# B&R Automation Studio project AGV
Automation Studio 4.7.3.93 SP

## Configuration CP1586

CPU X20CP1586, AutomationRuntime B4.91, Build 4.1.2, Vc V4.72.3

### Task classes (Cpu.sw)
```
Cyclic#1 (cycle 5000 us, tolerance 5000 us):
  motorCtrl <- ros_topics_typ.motorCtrl.prg
Binaries: FWRules, TCData, udbdef, User, iomap, Role, arconfig, asfw, ashwac, sysconf, ashwd, target, components
Libraries: ExOS, ExDeploy, ExData, runtime, sys_lib, FileIO, AsIOTime, ArEventLog, AsTCP, ros_topics, ROS, operator, astime, AsIecCon, brsystem, MTTypes, standard, MTFilter, MTBasics
```

### Hardware
```
X20CP1586 : X20CP1586 v1.9.0.0
  Connector IF2:
    ActivateDevice = 1
    Mode = Manual
    InternetAddress = 192.168.87.212
    SubnetMask = 255.255.255.0
  ConfigurationID = AGV_CP1586
  IdleTaskClass = 3
  TaskClassIdleTime = 2000
  Cyclic1Duration = 5000
  Cyclic1Tolerance = 5000
  Cyclic2Duration = 1000
  FileDevice1
  FileDeviceName1 = USER
  FileDevicePath1 = USER_PATH
  ActivateOpcUa = 1
  OpcUaInformationModels_PV_Version = 1
```

### target.exostarget - X20CP1586/exosTechnology/target.exostarget
```
Element gTarget_0 (Type=exostarget)
  General:
    ConnectionIP = 192.168.87.128
    Logging:
      LogLevel = Debug
      LogFilters:
        LogFilterUser = On
        LogFilterSystem = On
        LogFilterVerbose = On
      LogDestination = Volatile
    Deployment = On
      MaxRestarts = 10
    DataConnection = On
      ConnectionType = TCPIP
      TimeSynchronization:
        TimeConnection:
          TimePort = 49001
        PrecisionUsec = 1000
        GuardTimeSec = 36
        DeviationPerHourUsec = 100000
      DataConnectionLogging:
        LogConnection:
          LogPort = 49002
          LogShmPath = exos_log
        LogCycleTimeMsec = 50
  Components:
    ComponentsGeneral:
      ComponentsHeartbeatMsec = 500
      ComponentsTimeoutSec = 2
      ComponentsTaskClass = 2
      ComponentsCycleTimeMsec = 10
    Component[0]:
      ComponentConfigurationLink = gros_topics_typ_0
      DataModels:
        Instance[0]:
          InstanceName = ros_topics_typ_0
          InstanceConnection:
            InstancePort = 49003
            InstanceShmPath = ros_topics_typ_0
  ComponentDataConnection:
    Version = 2.0.0-1
    ErrorHandling = Target
    RestartEvent = Target
    StartupTimeout = 5
    Predefined:
      Files:
        File[0]:
          FileName = ufw-exos-data
          ChangeEvent = Ignore
        File[1]:
          FileName = exos-data-ports-allow.sh
          ChangeEvent = Restart
        File[2]:
          FileName = exos-data.conf
          ChangeEvent = Restart
        File[3]:
          FileName = exos-data_2.0.0-1_amd64.deb
          ChangeEvent = Reinstall
        File[4]:
          FileName = exos-data-eth_2.0.0-1_amd64.deb
          ChangeEvent = Reinstall
        File[5]:
          FileName = exos-data-remove.sh
          ChangeEvent = Ignore
        File[6]:
          FileName = run_server.sh
          ChangeEvent = Ignore
        File[7]:
          FileName = setup_build_environment.sh
          ChangeEvent = Ignore
        File[8]:
          FileName = libzmq5_4.2.1-4+deb9u2_amd64.deb
          ChangeEvent = Reinstall
        File[9]:
          FileName = libpgm-5.2-0_5.2.122~dfsg-2_amd64.deb
          ChangeEvent = Reinstall
        File[10]:
          FileName = libsodium18_1.0.11-2_amd64.deb
          ChangeEvent = Reinstall
      Services:
        Service[0]:
          Type = Install
          Command = dpkg -i *.deb
          WorkingDirectory
        Service[1]:
          Type = Remove
          Command = dpkg --purge exos-data
          WorkingDirectory
        Service[2]:
          Type = Remove
          Command = dpkg --purge exos-data-eth
          WorkingDirectory
        Service[3]:
          Type = Remove
          Command = sh exos-data-remove.sh
          WorkingDirectory
        Service[4]:
          Type = Startup
          Command = cp exos-data.conf /etc/exos-data.conf
          WorkingDirectory
        Service[5]:
          Type = Startup
          Command = cp ufw-exos-data /etc/ufw/applications.d/ufw-exos-data
          WorkingDirectory
        Service[6]:
          Type = Startup
          Command = sh exos-data-ports-allow.sh
          WorkingDirectory
        Service[7]:
          Type = Runtime
          Command = /usr/bin/exos_mr
          WorkingDirectory
  Simulation:
    SimConnectionIP = 192.168.87.128
    SimDeployment = On
    SimDataConnection = On
      SimConnectionType = TCPIP
      SimTimeSynchronization:
        SimPrecisionUsec = 5000
        SimGuardTimeSec = 30
    SimComponentsGeneral:
      SimComponentsHeartbeatMsec = 1000
      SimComponentsTimeoutSec = 75
```

## Configuration Config1

CPU X90CP174.48-00, AutomationRuntime C4.72, Build 4.1.2, Vc V4.72.0

### Task classes (Cpu.sw)
```
Cyclic#1 (cycle 5000 us, tolerance 0 us):
  motorCtrl <- motorCtrl.prg
Binaries: udbdef, FWRules, TCData, iomap, ashwac, Role, sysconf, arconfig, asfw, User, ashwd
Libraries: MTBasics, brsystem, MTTypes, sys_lib, runtime, asieccon, astime, MTFilter, ROS, standard
```

### Hardware
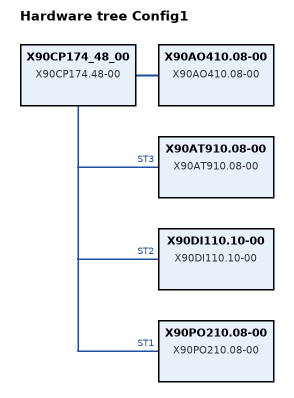
```
X90AO410.08-00 : X90AO410.08-00 v1.1.0.0  [ST -> X90CP174_48_00.ST4]
X90AT910.08-00 : X90AT910.08-00 v1.0.2.0  [ST -> X90CP174_48_00.ST3]
X90CP174_48_00 : X90CP174.48-00 v1.2.2.0  [X1 -> X1.SL]
  Module X1 (Type=X1, Virtual=true, Version=1.2.2.0)
    Connection (Connector=SL, TargetModule=X90CP174_48_00, TargetConnector=X1)
    ChannelConfig01 = 42
    DigitalFilterPin01 = 0
    ChannelConfig02 = 42
    DigitalFilterPin02 = 0
    ChannelConfig03 = 42
    DigitalFilterPin03 = 0
    ChannelConfig04 = 42
    DigitalFilterPin04 = 0
    IN1_CounterFunction01 = 3
    IN1_CounterFunction02 = 3
    ChannelConfig33 = 15
    PWMSource33 = 1
    PWMSyncPeriod33 = 125
    ChannelConfig34 = 20
    ChannelConfig35 = 20
    ChannelConfig36 = 20  // Configuration and impedance of pin X1.A.J1  
    ChannelConfig37 = 16
    ChannelConfig38 = 20  // Configuration and impedance of pin X1.A.L1  (6A)
    ChannelConfig39 = 20  // Configuration and impedance of pin X1.A.M2 (6A)
    ChannelConfig40 = 20
    ChannelConfig41 = 15
    PWMSource41 = 1
    PWMSyncPeriod41 = 125
    PWMDisplacement41 = 62
    ChannelConfig42 = 20
    ChannelConfig43 = 20  // Configuration and impedance of pin X1.B.H1  (6A)
    ChannelConfig44 = 20  // Configuration and impedance of pin X1.B.H3  (6A)
    ChannelConfig45 = 16  // Configuration and impedance of pin X1.B.G4  (6A)
    ChannelConfig46 = 20
    ChannelConfig47 = 20
    ChannelConfig48 = 20
  Connector IF2:
    ActivateDevice = 1
    Mode = Manual
    InternetAddress = 192.168.87.230
    SubnetMask = 255.255.255.0
  ConfigurationID = AGV_Config1
  EnableUsbRemoteInstall = 1
  EnableCfRemoteInstall = 1
  Cyclic1Duration = 5000
  Cyclic1Tolerance = 0
  Cyclic2Duration = 20000
  Cyclic2Tolerance = 20000
  Cyclic3Duration = 50000
  Cyclic3Tolerance = 50000
  Cyclic4Duration = 100000
  Cyclic4Tolerance = 100000
  Cyclic5Duration = 200000
  Cyclic5Tolerance = 200000
  Cyclic6Duration = 500000
  Cyclic6Tolerance = 500000
  Cyclic7Duration = 1000000
  Cyclic7Tolerance = 1000000
  Cyclic8Duration = 10000
  Cyclic8Tolerance = 30000000
  ActivateOpcUa = 1
  OpcUaInformationModels_PV_Version = 2
X90DI110.10-00 : X90DI110.10-00 v1.0.1.0  [ST -> X90CP174_48_00.ST2]
X90PO210.08-00 : X90PO210.08-00 v1.2.0.0  [ST -> X90CP174_48_00.ST1]
```

### IoMap.iom - X90CP174_48_00/IoMap.iom
```iecst
VAR_CONFIG
	::motorCtrl:localVariables[0].hw.output.pwm AT %QW."X1".PWMOutput33;
	::motorCtrl:localVariables[0].hw.input.encoder AT %IW."X1".Encoder01;
	::motorCtrl:localVariables[0].hw.input.current[0] AT %IW."X1".Current33;
	::motorCtrl:localVariables[0].hw.input.current[1] AT %IW."X1".Current34;
	::motorCtrl:localVariables[0].hw.input.current[2] AT %IW."X1".Current35;
	::motorCtrl:localVariables[0].hw.input.current[3] AT %IW."X1".Current36;
	::motorCtrl:localVariables[0].hw.input.overload AT %IX."X1".OverloadDigitalOutput33;
	::motorCtrl:localVariables[0].hw.output.clear AT %QX."X1".OverloadClear33;
	::motorCtrl:localVariables[1].hw.input.encoder AT %IW."X1".Encoder02;
	::motorCtrl:localVariables[1].hw.output.pwm AT %QW."X1".PWMOutput37;
	::motorCtrl:localVariables[0].hw.input.current[4] AT %IW."X1".Current37;
	::motorCtrl:localVariables[0].hw.input.current[6] AT %IW."X1".Current39;
	::motorCtrl:localVariables[1].hw.input.nettime AT %ID."X90CP174_48_00".SystemTime;
	::motorCtrl:localVariables[0].hw.input.nettime AT %ID."X90CP174_48_00".SystemTime;
	::motorCtrl:localVariables[0].hw.input.current[5] AT %IW."X1".Current38;
	::motorCtrl:localVariables[0].hw.input.current[7] AT %IW."X1".Current40;
	::motorCtrl:localVariables[1].hw.output.pwm AT %QW."X1".PWMOutput41;
	::motorCtrl:localVariables[1].hw.output.clear AT %QX."X1".OverloadClear41;
	::motorCtrl:localVariables[1].hw.input.current[0] AT %IW."X1".Current41;
	::motorCtrl:localVariables[1].hw.input.overload  AT %IX."X1".OverloadDigitalOutput41;
	::motorCtrl:localVariables[1].hw.input.current[1]  AT %IW."X1".Current42;
	::motorCtrl:localVariables[1].hw.input.current[2]  AT %IW."X1".Current43;
	::motorCtrl:localVariables[1].hw.input.current[3]  AT %IW."X1".Current44;
	::motorCtrl:localVariables[1].hw.input.current[4]  AT %IW."X1".Current45;
	::motorCtrl:localVariables[1].hw.input.current[5]  AT %IW."X1".Current46;
	::motorCtrl:localVariables[1].hw.input.current[6]  AT %IW."X1".Current47;
	::motorCtrl:localVariables[1].hw.input.current[7]  AT %IW."X1".Current48;
END_VAR
```

### components.exoscomponent - X90CP174_48_00/exosTechnology/components.exoscomponent
```
Element gros_topics_typ_0 (Type=exoscomponent)
  PackageSelection = Logical\ros_topics_typ\ros_topics_typ.exospkg
  ErrorHandling = Component
  RestartEvent = Component
  StartupTimeout = 0
  Predefined:
    Files:
      File[0]:
        FileName = Linux\ros_topics_typ.py
        ChangeEvent = Restart
      File[1]:
        FileName = Linux\exos-comp-ros_topics_typ_1.0.0_amd64.deb
        ChangeEvent = Reinstall
    Services:
      Service[0]:
        Type = Install
        Command = dpkg -i exos-comp-ros_topics_typ_1.0.0_amd64.deb
        WorkingDirectory
      Service[1]:
        Type = Remove
        Command = dpkg --purge exos-comp-ros_topics_typ
        WorkingDirectory
      Service[2]:
        Type = Startup
        Command = cp ros_topics_typ.py /home/user/brdkAGV_linux/ros_ws/src/motor_control_exos/motor_control_exos/motor_control_exos.py
        WorkingDirectory
Element gWaterTank_0 (Type=exoscomponent)
  PackageSelection = Logical\WaterTank\WaterTank.exospkg
  ErrorHandling = Component
  RestartEvent = Component
  StartupTimeout = 0
  Predefined:
    Files:
      File[0]:
        FileName = Linux\watertank.py
        ChangeEvent = Restart
      File[1]:
        FileName = Linux\exos-comp-watertank_1.0.0_amd64.deb
        ChangeEvent = Reinstall
    Services:
      Service[0]:
        Type = Install
        Command = dpkg -i exos-comp-watertank_1.0.0_amd64.deb
        WorkingDirectory
      Service[1]:
        Type = Remove
        Command = dpkg --purge exos-comp-watertank
        WorkingDirectory
      Service[2]:
        Type = Startup
        Command = cp watertank.py /home/user/watertank
        WorkingDirectory
      Service[3]:
        Type = Runtime
        Command = python3 watertank.py
        WorkingDirectory = /home/user/watertank
```

### target.exostarget - X90CP174_48_00/exosTechnology/target.exostarget
```
Element gTarget_0 (Type=exostarget)
  General:
    ConnectionIP = 192.168.87.128
    Logging:
      LogLevel = Debug
      LogFilters:
        LogFilterUser = On
        LogFilterSystem = On
        LogFilterVerbose = On
      LogDestination = Volatile
    Deployment = On
      MaxRestarts = 10
    DataConnection = On
      ConnectionType = TCPIP
      TimeSynchronization:
        TimeConnection:
          TimePort = 49001
        PrecisionUsec = 5000
        GuardTimeSec = 180
        DeviationPerHourUsec = 100000
      DataConnectionLogging:
        LogConnection:
          LogPort = 49002
          LogShmPath = exos_log
        LogCycleTimeMsec = 50
  Components:
    ComponentsGeneral:
      ComponentsHeartbeatMsec = 500
      ComponentsTimeoutSec = 2
      ComponentsTaskClass = 2
      ComponentsCycleTimeMsec = 10
    Component[0]:
      ComponentConfigurationLink = gros_topics_typ_0
      DataModels:
        Instance[0]:
          InstanceName = ros_topics_typ_0
          InstanceConnection:
            InstancePort = 49003
            InstanceShmPath = ros_topics_typ_0
    Component[1]:
      ComponentConfigurationLink = gWaterTank_0
      DataModels:
        Instance[0]:
          InstanceName = WaterTank_0
          InstanceConnection:
            InstancePort = 49004
            InstanceShmPath = WaterTank_0
  ComponentDataConnection:
    Version = 2.1.0-1
    ErrorHandling = Target
    RestartEvent = Target
    StartupTimeout = 5
    Predefined:
      Files:
        File[0]:
          FileName = ufw-exos-data
          ChangeEvent = Ignore
        File[1]:
          FileName = exos-data-ufw-profile.sh
          ChangeEvent = Ignore
        File[2]:
          FileName = exos-data-ports-allow.sh
          ChangeEvent = Restart
        File[3]:
          FileName = exos-data.conf
          ChangeEvent = Restart
        File[4]:
          FileName = exos-data_2.1.0-1_amd64.deb
          ChangeEvent = Reinstall
        File[5]:
          FileName = exos-data-eth_2.1.0-1_amd64.deb
          ChangeEvent = Reinstall
        File[6]:
          FileName = exos-data-remove.sh
          ChangeEvent = Ignore
        File[7]:
          FileName = run_server.sh
          ChangeEvent = Ignore
        File[8]:
          FileName = setup_build_environment.sh
          ChangeEvent = Ignore
        File[9]:
          FileName = libzmq5_4.2.1-4+deb9u2_amd64.deb
          ChangeEvent = Reinstall
        File[10]:
          FileName = libpgm-5.2-0_5.2.122~dfsg-2_amd64.deb
          ChangeEvent = Reinstall
        File[11]:
          FileName = libsodium18_1.0.11-2_amd64.deb
          ChangeEvent = Reinstall
      Services:
        Service[0]:
          Type = Install
          Command = dpkg -i *.deb
          WorkingDirectory
        Service[1]:
          Type = Remove
          Command = dpkg --purge exos-data
          WorkingDirectory
        Service[2]:
          Type = Remove
          Command = dpkg --purge exos-data-eth
          WorkingDirectory
        Service[3]:
          Type = Remove
          Command = sh exos-data-remove.sh
          WorkingDirectory
        Service[4]:
          Type = Startup
          Command = cp exos-data.conf /etc/exos-data.conf
          WorkingDirectory
        Service[5]:
          Type = Startup
          Command = sh exos-data-ufw-profile.sh
          WorkingDirectory
        Service[6]:
          Type = Startup
          Command = sh exos-data-ports-allow.sh
          WorkingDirectory
        Service[7]:
          Type = Runtime
          Command = /usr/bin/exos_mr
          WorkingDirectory
  Simulation:
    SimConnectionIP = 192.168.87.128
    SimDeployment = On
    SimDataConnection = On
      SimConnectionType = TCPIP
      SimTimeSynchronization:
        SimPrecisionUsec = 10000
        SimGuardTimeSec = 30
    SimComponentsGeneral:
      SimComponentsHeartbeatMsec = 1000
      SimComponentsTimeoutSec = 75
```

## Logical view

Binary libraries used (declarations not repeated): operator, runtime, astime, AsIecCon, MTBasics 5.06.0, brsystem, MTTypes, sys_lib, MTFilter 5.06.0, standard, AsIOTime, ExOS 2.01.0

### Package Logical/Libraries - Global libraries

### Library Logical/Libraries/ROS (ANSIC)

#### Types.typ - Exported data types
```iecst
TYPE
	ros_topic_point_typ : 	STRUCT  (*this expresses velocity in free space broken into its linear and angular parts.*)
		y : LREAL;
		z : LREAL;
		x : LREAL;
	END_STRUCT;
	ros_topic_vector3_typ : 	STRUCT  (*this expresses velocity in free space broken into its linear and angular parts.*)
		y : LREAL;
		z : LREAL;
		x : LREAL;
	END_STRUCT;
	ros_topic_twist_typ : 	STRUCT  (*This expresses velocity in free space broken into its linear and angular parts.*)
		angular : ros_topic_vector3_typ;
		linear : ros_topic_vector3_typ;
	END_STRUCT;
	ros_topic_twistCor_typ : 	STRUCT  (*This expresses velocity in free space with uncertainty.*)
		twist : ros_topic_twist_typ;
		covariance : ARRAY[0..63]OF LREAL; (*Row-major representation of the 6x6 covariance matrix
The orientation parameters use a fixed-axis representation. In order, the parameters are:
 (x, y, z, rotation about X axis, rotation about Y axis, rotation about Z axis)*)
	END_STRUCT;
	ros_topic_quaternion_typ : 	STRUCT  (*This represents an orientation in free space in quaternion form.*)
		y : LREAL;
		z : LREAL;
		w : LREAL;
		x : LREAL;
	END_STRUCT;
	ros_topic_odemety_point_typ : 	STRUCT  (*This contains the position of a point in free space*)
		y : LREAL;
		z : LREAL;
		x : LREAL;
	END_STRUCT;
	ros_topic_pose_typ : 	STRUCT  (*A representation of pose in free space, composed of position and orientation. *)
		position : ros_topic_point_typ;
		orientation : ros_topic_quaternion_typ;
	END_STRUCT;
	ros_topic_poseCor_typ : 	STRUCT  (*This represents a pose in free space with uncertainty.*)
		pose : ros_topic_pose_typ;
		covariance : ARRAY[0..63]OF LREAL; (*Row-major representation of the 6x6 covariance matrix
The orientation parameters use a fixed-axis representation. In order, the parameters are:
 (x, y, z, rotation about X axis, rotation about Y axis, rotation about Z axis)*)
	END_STRUCT;
	ros_topic_time_typ : 	STRUCT
		nsec : UDINT;
		sec : UDINT;
	END_STRUCT;
	ros_topic_header_typ : 	STRUCT
		stamp : ros_topic_time_typ;
		seq : UDINT;
		frame_id : STRING[20];
	END_STRUCT;
	ros_topic_odemety_typ : 	STRUCT
		pose : ros_topic_poseCor_typ;
		twist : ros_topic_twistCor_typ;
		header : ros_topic_header_typ;
	END_STRUCT;
END_TYPE
```

#### ROS.fun - Exported functions and function blocks
```iecst
{REDUND_ERROR} FUNCTION normalizeAngle : LREAL (*TODO: Add your comment here*) (*$GROUP=User,$CAT=User,$GROUPICON=User.png,$CATICON=User.png*)
	VAR_INPUT
		angle : LREAL;
	END_VAR
END_FUNCTION
```

#### normalizeAngle.c
```c
#include <bur/plctypes.h>
#ifdef __cplusplus
	extern "C"
	{
#endif
	#include "ROS.h"
#ifdef __cplusplus
	};
#endif

#define M_PI 3.14159265358979323846

/* TODO: Add your comment here */
double normalizeAngle(double angle)
{

	if( angle > M_PI){
		angle -= 2.0 * M_PI;
	}
	if(angle < -M_PI){
		angle += 2.0 * M_PI;
	}

	return angle;
}
```

### Program Logical/motorCtrl (IEC)

#### Main.st - Init, cyclic, exit code
```iecst
PROGRAM _INIT
	(* Insert code here *)
	FOR i:=0 TO i < 2 BY 1 DO
		setupPointers;

		this.PID.Enable := TRUE;
		this.PID.MinOut := -100;
		this.PID.MaxOut := 100;
		this.PID.PIDParameters.DerivativeTime := 0.00228000456;
		this.PID.PIDParameters.Gain := 78;
		this.PID.PIDParameters.IntegrationTime := 0.02500019;
		this.PID.PIDParameters.FilterTime := 0.000228000456;

		this.PID.Update := TRUE;

		this.PIDCurrent.Enable := TRUE;
		this.PIDCurrent.MinOut := 0;
		this.PIDCurrent.MaxOut := 100;
		this.PIDCurrent.PIDParameters.DerivativeTime := 10;
		this.PIDCurrent.PIDParameters.Gain := 1;
		this.PIDCurrent.PIDParameters.IntegrationTime := 10;
		this.PIDCurrent.PIDParameters.FilterTime := 20;
		this.PIDCurrent.Update := TRUE;
		this.PIDCurrent.SetValue := 8;

		this.filterSpeed.Enable := TRUE;
		this.filterSpeed.WindowLength := 100;
		this.filterSpeed.Update := TRUE;

		this.filterCurrent.Enable := TRUE;
		this.filterCurrent.WindowLength := 3;
		this.filterCurrent.Update := TRUE;

		this.accLimiter.Enable := TRUE;
		this.accLimiter.MaxNegSlewRate := 1;
		this.accLimiter.MaxPosSlewRate := 1;
		this.accLimiter.MaxOut := 2;
		this.accLimiter.MinOut := -2;
		this.accLimiter.Update := TRUE;

		this.PIDtune.SetValue:= 1.0;
		this.PIDtune.MinOut:= 0.0;
		this.PIDtune.MaxOut:= 100.0;
		this.PIDtune.Update := TRUE;

		this.lowPass.Enable := TRUE;
		this.lowPass.CutOffFrequency := 10;
		this.lowPass.Order := 1;
		this.lowPass.Update := TRUE;

		this.encoderOld := this.hw.input.encoder;
		this.timeOld := this.hw.input.nettime;

		this.ton_overcurrent.PT := T#1s;

	END_FOR

END_PROGRAM

PROGRAM _CYCLIC
	(* Insert code here *)

	ros.topics.twist.linear.x := MAX(MIN(ros.topics.twist.linear.x,ros.topics.config.maxSpeed),ros.topics.config.minSpeed);

	IF localVariables[0].hmi.output.overload OR localVariables[1].hmi.output.overload  THEN
		localVariables[0].PID.SetValue := 0;
		localVariables[1].PID.SetValue := 0;
	ELSE
		localVariables[0].PID.SetValue := LREAL_TO_REAL(ros.topics.twist.linear.x + ros.topics.twist.angular.z * ros.topics.config.baseWidth / 2.0) * ros.currentLimiter;  // m/s
		localVariables[1].PID.SetValue := LREAL_TO_REAL(ros.topics.twist.linear.x - ros.topics.twist.angular.z * ros.topics.config.baseWidth / 2.0) * ros.currentLimiter;
	END_IF

	FOR i:=0 TO 1 BY 1 DO
		setupPointers;

		hmi.output.overload := FALSE;

		hmi.output.currentTotal := 0;

		FOR k:=0 TO 7 DO

			hmi.output.current[k] := INT_TO_REAL(hw.input.current[k])*10.0/32767.0;
			hmi.output.currentTotal := hmi.output.currentTotal + hmi.output.current[k];
		END_FOR

		hmi.output.currentTotal := hmi.output.currentTotal /2.0;

		IF this.filterCurrent.UpdateDone THEN
			this.filterSpeed.Update := FALSE;
		END_IF

		this.filterCurrent(In := hmi.output.currentTotal);

		IF this.PIDCurrent.UpdateDone THEN
			this.PIDCurrent.Update := FALSE;
		END_IF

		this.PIDCurrent(ActValue := this.filterCurrent.Out);

		this.currentLimiter := 1;//this.PIDCurrent.Out/100;

		hmi.output.overload := hw.input.overload;

		this.ton_overcurrent(IN := hmi.output.overload);
		IF this.ton_overcurrent.Q THEN
			this.hmi.input.clear := TRUE;
		END_IF

		hw.output.clear := hmi.input.clear;

		IF NOT hmi.output.overload THEN
			hmi.input.clear := FALSE;
		END_IF

		this.diffTime := DINT_TO_LREAL(hw.input.nettime -this.timeOld);
		IF this.diffTime < -100000.0 THEN
			this.diffTime := this.diffTime + 2*2147483647;
		END_IF
		this.diffTime := this.diffTime /1000.0;
		this.timeOld := hw.input.nettime;

		this.diffEncoder := INT_TO_LREAL(hw.input.encoder)-INT_TO_LREAL(this.encoderOld);

		this.encoderOld := hw.input.encoder;

		IF this.diffEncoder > 32727 THEN

			this.diffEncoder := this.diffEncoder - 2*32767;

		ELSIF this.diffEncoder < -32727 THEN

			this.diffEncoder := this.diffEncoder + 2*32767;

		END_IF

		hmi.output.ticks := hmi.output.ticks + this.diffEncoder;
		hmi.output.distance := hmi.output.ticks / UDINT_TO_LREAL(config.ppm);

		IF hmi.input.resetDistance THEN
			hmi.input.resetDistance := FALSE;
			hmi.output.ticks := 0;
			hmi.output.distance := 0;
		END_IF

		this.distance 	:= this.diffEncoder/UDINT_TO_LREAL(config.ppm);

		this.lowPass.In := LREAL_TO_REAL(this.distance);
		this.lowPass();

		this.speed 		:= this.distance * 1000/this.diffTime;

		IF this.filterSpeed.UpdateDone THEN
			this.filterSpeed.Update := FALSE;
		END_IF

		this.filterSpeed(In := LREAL_TO_REAL(this.speed));

		IF this.accLimiter.UpdateDone THEN
			this.accLimiter.Update := FALSE;
		END_IF

		this.accLimiter(In := this.PID.SetValue);

		IF this.PID.UpdateDone THEN
			this.PID.Update := FALSE;
		END_IF

		this.PID.ActValue := LREAL_TO_REAL(this.speed);
		this.PID.SetValue := this.accLimiter.Out;
		// PID TUNE

		IF hmi.input.tune THEN
			this.PIDtune.Enable := TRUE;
		END_IF

		this.PIDtune.ActValue := LREAL_TO_REAL(this.speed);

		IF this.PIDtune.TuningDone THEN
			this.PIDtune.Start := FALSE;
			this.PID.IntegrationPartPresetValue := this.PIDtune.Out;
			this.PID.SetIntegrationPart := TRUE;
		ELSIF this.PIDtune.Active AND NOT this.PIDtune.Update THEN
			//	this.PIDtune.Start := TRUE;
		END_IF

		IF this.PIDtune.UpdateDone THEN
			this.PIDtune.Update := FALSE;
		END_IF

		(* call function block *)
		this.PID();
		this.PIDtune();

		this.PID.SetIntegrationPart := FALSE;

		IF hmi.input.tune THEN
			hw.output.pwm := REAL_TO_INT(this.PIDtune.Out*327.67);
		ELSE
			hw.output.pwm := REAL_TO_INT(this.PID.Out*327.67);
		END_IF

	END_FOR

	ros.currentLimiter := MIN(localVariables[0].currentLimiter,localVariables[1].currentLimiter);

	ros.diffDist := localVariables[1].distance-localVariables[0].distance;
	ros.diffLowpassDist := localVariables[1].lowPass.Out-localVariables[0].lowPass.Out;

	ros.dist := (localVariables[1].distance+localVariables[0].distance)/2;

	IF localVariables[0].diffEncoder = localVariables[1].diffEncoder THEN
		ros.d_theta := 0.0;
		ros.cur_x := ros.cur_x + ros.dist * COS(ros.cur_theta);
		ros.cur_y := ros.cur_y + ros.dist * SIN(ros.cur_theta);
	ELSE
		ros.d_theta := (localVariables[1].distance - localVariables[0].distance) / ros.topics.config.baseWidth;
		ros.dist := (localVariables[1].distance+localVariables[0].distance)/2;
		ros.r := ros.dist / ros.d_theta;
		ros.cur_x := ros.cur_x + ros.r * (SIN(ros.d_theta + ros.cur_theta) - SIN(ros.cur_theta));
		ros.cur_y := ros.cur_y - ros.r * (COS(ros.d_theta + ros.cur_theta) - COS(ros.cur_theta));
		ros.cur_theta := normalizeAngle(ros.cur_theta + ros.d_theta);
	END_IF

	ros.vel_x := ros.dist * (1000.0/localVariables[0].diffTime);
	ros.vel_theta := ros.d_theta * (1000.0/localVariables[0].diffTime);

	// set ros data
	ros.topics.odemetry.pose.pose.position.x 	:= ros.cur_x;
	ros.topics.odemetry.pose.pose.position.y	:= ros.cur_y;
	ros.topics.odemetry.pose.pose.orientation.z	:= ros.cur_theta;

	ros.topics.odemetry.twist.twist.linear.x  	:= ros.vel_x;
	ros.topics.odemetry.twist.twist.angular.z 	:= ros.vel_theta;

	setupWatchPointers;

END_PROGRAM

PROGRAM _EXIT
	(* Insert code here *)

END_PROGRAM
```

#### Types.typ - Local data types
```iecst
TYPE
	ros_config_typ : 	STRUCT
		maxSpeed : LREAL := 2;
		minSpeed : LREAL := -2;
		baseWidth : LREAL := 0.53;
	END_STRUCT;
	ros_topics_typ : 	STRUCT
		odemetry : ros_topic_odemety_typ;
		twist : ros_topic_twist_typ;
		config : ros_config_typ;
	END_STRUCT;
	ros_typ : 	STRUCT
		vel_theta : LREAL;
		vel_x : LREAL;
		r : LREAL;
		cur_theta : LREAL;
		dist : LREAL;
		cur_y : LREAL;
		cur_x : LREAL;
		d_theta : LREAL;
		topics : ros_topics_typ;
		diffLowpassDist : REAL;
		diffDist : LREAL;
		currentLimiter : REAL;
	END_STRUCT;
	local_typ : 	STRUCT
		hw : hw_typ;
		hmi : hmi_typ;
		speed : LREAL;
		encoderOld : INT;
		accLimiter : MTBasicsLimiter;
		PIDCurrent : MTBasicsPID;
		PID : MTBasicsPID;
		distance : LREAL;
		diffEncoder : LREAL;
		filterCurrent : MTFilterMovingAverage;
		filterSpeed : MTFilterMovingAverage;
		diffTime : LREAL;
		timeOld : DINT;
		PIDtune : MTBasicsOscillationTuning;
		lowPass : MTFilterLowPass;
		ton_overcurrent : TON;
		currentLimiter : REAL;
	END_STRUCT;
	hw_typ : 	STRUCT
		input : hw_input_typ;
		output : hw_output_typ;
	END_STRUCT;
	hw_output_typ : 	STRUCT
		pwm : INT;
		clear : BOOL;
	END_STRUCT;
	hw_input_typ : 	STRUCT
		encoder : INT;
		overload : BOOL;
		current : ARRAY[0..7]OF INT;
		nettime : DINT;
	END_STRUCT;
	hmi_typ : 	STRUCT
		config : config_typ;
		output : hmi_output_typ;
		input : hmi_input_typ;
	END_STRUCT;
	hmi_output_typ : 	STRUCT
		current : ARRAY[0..7]OF REAL;
		overload : BOOL;
		distance : LREAL;
		ticks : LREAL;
		currentTotal : REAL;
	END_STRUCT;
	hmi_input_typ : 	STRUCT
		clear : BOOL;
		tune : BOOL;
		resetDistance : BOOL;
	END_STRUCT;
	config_typ : 	STRUCT
		ppm : UDINT := 105860;
		maxCurrent : REAL := 8;
	END_STRUCT;
	common_typ : 	STRUCT
	END_STRUCT;
END_TYPE
```

#### Variables.var - Local variables
```iecst
VAR
	ros : ros_typ;
	config : REFERENCE TO config_typ;
	hmi : REFERENCE TO hmi_typ;
	hw : REFERENCE TO hw_typ;
	this : REFERENCE TO local_typ;
	localVariables : ARRAY[0..1] OF local_typ;
	watchIdx : USINT;
	k : USINT;
	i : USINT;
END_VAR
```

- ros_topics_typ.exospkg (not shown)

### libros_topics_typ.c - ros_topics_typ static library wrapper source
```c
#include <string.h>
#define EXOS_ASSERT_LOG &logger
#include "exos_log.h"
#include "libros_topics_typ.h"

#define SUCCESS(_format_, ...) exos_log_success(&logger, EXOS_LOG_TYPE_USER, _format_, ##__VA_ARGS__);
#define INFO(_format_, ...) exos_log_info(&logger, EXOS_LOG_TYPE_USER, _format_, ##__VA_ARGS__);
#define VERBOSE(_format_, ...) exos_log_debug(&logger, EXOS_LOG_TYPE_USER + EXOS_LOG_TYPE_VERBOSE, _format_, ##__VA_ARGS__);
#define ERROR(_format_, ...) exos_log_error(&logger, _format_, ##__VA_ARGS__);

static exos_log_handle_t logger;

typedef struct libros_topics_typHandle
{
    libros_topics_typ_t ext_ros_topics_typ_datamodel;
    exos_datamodel_handle_t ros_topics_typ_datamodel;

    exos_dataset_handle_t odemetry_dataset;
    exos_dataset_handle_t twist_dataset;
    exos_dataset_handle_t config_dataset;
} libros_topics_typHandle_t;

static libros_topics_typHandle_t h_ros_topics_typ;

static void libros_topics_typ_datasetEvent(exos_dataset_handle_t *dataset, EXOS_DATASET_EVENT_TYPE event_type, void *info)
{
    switch (event_type)
    {
    case EXOS_DATASET_EVENT_UPDATED:
        VERBOSE("dataset %s updated! latency (us):%i", dataset->name, (exos_datamodel_get_nettime(dataset->datamodel) - dataset->nettime));
        //handle each subscription dataset separately
        if (0 == strcmp(dataset->name, "odemetry"))
        {
            //update the nettime
            h_ros_topics_typ.ext_ros_topics_typ_datamodel.odemetry.nettime = dataset->nettime;

            //trigger the callback if assigned
            if (NULL != h_ros_topics_typ.ext_ros_topics_typ_datamodel.odemetry.on_change)
            {
                h_ros_topics_typ.ext_ros_topics_typ_datamodel.odemetry.on_change();
            }
        }
        break;

    default:
        break;
    }
}

static void libros_topics_typ_datamodelEvent(exos_datamodel_handle_t *datamodel, const EXOS_DATAMODEL_EVENT_TYPE event_type, void *info)
{
    switch (event_type)
    {
    case EXOS_DATAMODEL_EVENT_CONNECTION_CHANGED:
        INFO("application changed state to %s", exos_get_state_string(datamodel->connection_state));

        h_ros_topics_typ.ext_ros_topics_typ_datamodel.is_connected = false;
        h_ros_topics_typ.ext_ros_topics_typ_datamodel.is_operational = false;
        switch (datamodel->connection_state)
        {
        case EXOS_STATE_DISCONNECTED:
            if (NULL != h_ros_topics_typ.ext_ros_topics_typ_datamodel.on_disconnected)
            {
                h_ros_topics_typ.ext_ros_topics_typ_datamodel.on_disconnected();
            }
            break;
        case EXOS_STATE_CONNECTED:
            h_ros_topics_typ.ext_ros_topics_typ_datamodel.is_connected = true;
            if (NULL != h_ros_topics_typ.ext_ros_topics_typ_datamodel.on_connected)
            {
                h_ros_topics_typ.ext_ros_topics_typ_datamodel.on_connected();
            }
            break;
        case EXOS_STATE_OPERATIONAL:
            h_ros_topics_typ.ext_ros_topics_typ_datamodel.is_connected = true;
            h_ros_topics_typ.ext_ros_topics_typ_datamodel.is_operational = true;
            if (NULL != h_ros_topics_typ.ext_ros_topics_typ_datamodel.on_operational)
            {
                h_ros_topics_typ.ext_ros_topics_typ_datamodel.on_operational();
            }
            SUCCESS("ros_topics_typ operational!");
            break;
        case EXOS_STATE_ABORTED:
            if (NULL != h_ros_topics_typ.ext_ros_topics_typ_datamodel.on_disconnected)
            {
                h_ros_topics_typ.ext_ros_topics_typ_datamodel.on_disconnected();
            }
            ERROR("application error %d (%s) occured", datamodel->error, exos_get_error_string(datamodel->error));
            break;
        }
        break;
    case EXOS_DATAMODEL_EVENT_SYNC_STATE_CHANGED:
        break;

    default:
        break;

    }
}

static void libros_topics_typ_publish_twist_dataset(void)
{
    exos_dataset_publish(&h_ros_topics_typ.twist_dataset);
}
static void libros_topics_typ_publish_config_dataset(void)
{
    exos_dataset_publish(&h_ros_topics_typ.config_dataset);
}

static void libros_topics_typ_connect(void)
{
    //connect the datamodel
    EXOS_ASSERT_OK(exos_datamodel_connect_ros_topics_typ(&(h_ros_topics_typ.ros_topics_typ_datamodel), libros_topics_typ_datamodelEvent));

    //connect datasets
    EXOS_ASSERT_OK(exos_dataset_connect(&(h_ros_topics_typ.odemetry_dataset), EXOS_DATASET_SUBSCRIBE, libros_topics_typ_datasetEvent));
    EXOS_ASSERT_OK(exos_dataset_connect(&(h_ros_topics_typ.twist_dataset), EXOS_DATASET_PUBLISH, libros_topics_typ_datasetEvent));
    EXOS_ASSERT_OK(exos_dataset_connect(&(h_ros_topics_typ.config_dataset), EXOS_DATASET_PUBLISH, libros_topics_typ_datasetEvent));
}
static void libros_topics_typ_disconnect(void)
{
    h_ros_topics_typ.ext_ros_topics_typ_datamodel.is_connected = false;
    h_ros_topics_typ.ext_ros_topics_typ_datamodel.is_operational = false;

    EXOS_ASSERT_OK(exos_datamodel_disconnect(&(h_ros_topics_typ.ros_topics_typ_datamodel)));
}

static void libros_topics_typ_set_operational(void)
{
    EXOS_ASSERT_OK(exos_datamodel_set_operational(&(h_ros_topics_typ.ros_topics_typ_datamodel)));
}

static void libros_topics_typ_process(void)
{
    EXOS_ASSERT_OK(exos_datamodel_process(&(h_ros_topics_typ.ros_topics_typ_datamodel)));
    exos_log_process(&logger);
}

static void libros_topics_typ_dispose(void)
{
    h_ros_topics_typ.ext_ros_topics_typ_datamodel.is_connected = false;
    h_ros_topics_typ.ext_ros_topics_typ_datamodel.is_operational = false;

    EXOS_ASSERT_OK(exos_datamodel_delete(&(h_ros_topics_typ.ros_topics_typ_datamodel)));
    exos_log_delete(&logger);
}

static int32_t libros_topics_typ_get_nettime(void)
{
    return exos_datamodel_get_nettime(&(h_ros_topics_typ.ros_topics_typ_datamodel));
}

static void libros_topics_typ_log_error(char* log_entry)
{
    exos_log_error(&logger, log_entry);
}

static void libros_topics_typ_log_warning(char* log_entry)
{
    exos_log_warning(&logger, EXOS_LOG_TYPE_USER, log_entry);
}

static void libros_topics_typ_log_success(char* log_entry)
{
    exos_log_success(&logger, EXOS_LOG_TYPE_USER, log_entry);
}

static void libros_topics_typ_log_info(char* log_entry)
{
    exos_log_info(&logger, EXOS_LOG_TYPE_USER, log_entry);
}

static void libros_topics_typ_log_debug(char* log_entry)
{
    exos_log_debug(&logger, EXOS_LOG_TYPE_USER, log_entry);
}

static void libros_topics_typ_log_verbose(char* log_entry)
{
    exos_log_warning(&logger, EXOS_LOG_TYPE_USER + EXOS_LOG_TYPE_VERBOSE, log_entry);
}

libros_topics_typ_t *libros_topics_typ_init(void)
{
    memset(&h_ros_topics_typ, 0, sizeof(h_ros_topics_typ));

    h_ros_topics_typ.ext_ros_topics_typ_datamodel.twist.publish = libros_topics_typ_publish_twist_dataset;
    h_ros_topics_typ.ext_ros_topics_typ_datamodel.config.publish = libros_topics_typ_publish_config_dataset;

    h_ros_topics_typ.ext_ros_topics_typ_datamodel.connect = libros_topics_typ_connect;
    h_ros_topics_typ.ext_ros_topics_typ_datamodel.disconnect = libros_topics_typ_disconnect;
    h_ros_topics_typ.ext_ros_topics_typ_datamodel.process = libros_topics_typ_process;
    h_ros_topics_typ.ext_ros_topics_typ_datamodel.set_operational = libros_topics_typ_set_operational;
    h_ros_topics_typ.ext_ros_topics_typ_datamodel.dispose = libros_topics_typ_dispose;
    h_ros_topics_typ.ext_ros_topics_typ_datamodel.get_nettime = libros_topics_typ_get_nettime;
    h_ros_topics_typ.ext_ros_topics_typ_datamodel.log.error = libros_topics_typ_log_error;
    h_ros_topics_typ.ext_ros_topics_typ_datamodel.log.warning = libros_topics_typ_log_warning;
    h_ros_topics_typ.ext_ros_topics_typ_datamodel.log.success = libros_topics_typ_log_success;
    h_ros_topics_typ.ext_ros_topics_typ_datamodel.log.info = libros_topics_typ_log_info;
    h_ros_topics_typ.ext_ros_topics_typ_datamodel.log.debug = libros_topics_typ_log_debug;
    h_ros_topics_typ.ext_ros_topics_typ_datamodel.log.verbose = libros_topics_typ_log_verbose;

    exos_log_init(&logger, "gros_topics_typ_0");

    SUCCESS("starting gros_topics_typ_0 application..");

    EXOS_ASSERT_OK(exos_datamodel_init(&h_ros_topics_typ.ros_topics_typ_datamodel, "ros_topics_typ_0", "gros_topics_typ_0"));

    //set the user_context to access custom data in the callbacks
    h_ros_topics_typ.ros_topics_typ_datamodel.user_context = NULL; //not used
    h_ros_topics_typ.ros_topics_typ_datamodel.user_tag = 0; //not used

    EXOS_ASSERT_OK(exos_dataset_init(&h_ros_topics_typ.odemetry_dataset, &h_ros_topics_typ.ros_topics_typ_datamodel, "odemetry", &h_ros_topics_typ.ext_ros_topics_typ_datamodel.odemetry.value, sizeof(h_ros_topics_typ.ext_ros_topics_typ_datamodel.odemetry.value)));
    h_ros_topics_typ.odemetry_dataset.user_context = NULL; //not used
    h_ros_topics_typ.odemetry_dataset.user_tag = 0; //not used

    EXOS_ASSERT_OK(exos_dataset_init(&h_ros_topics_typ.twist_dataset, &h_ros_topics_typ.ros_topics_typ_datamodel, "twist", &h_ros_topics_typ.ext_ros_topics_typ_datamodel.twist.value, sizeof(h_ros_topics_typ.ext_ros_topics_typ_datamodel.twist.value)));
    h_ros_topics_typ.twist_dataset.user_context = NULL; //not used
    h_ros_topics_typ.twist_dataset.user_tag = 0; //not used

    EXOS_ASSERT_OK(exos_dataset_init(&h_ros_topics_typ.config_dataset, &h_ros_topics_typ.ros_topics_typ_datamodel, "config", &h_ros_topics_typ.ext_ros_topics_typ_datamodel.config.value, sizeof(h_ros_topics_typ.ext_ros_topics_typ_datamodel.config.value)));
    h_ros_topics_typ.config_dataset.user_context = NULL; //not used
    h_ros_topics_typ.config_dataset.user_tag = 0; //not used

    return &(h_ros_topics_typ.ext_ros_topics_typ_datamodel);
}
```

### CMakeLists.txt - CMake build file script
```
cmake_minimum_required(VERSION 3.0)

project(ros_topics_typ)

set(CMAKE_BUILD_TYPE Debug)
find_package(SWIG REQUIRED)
include(${SWIG_USE_FILE})

# Load Python Libraries
# ---------------------
# a.) use Python 3
find_package(PythonLibs 3)
# b.) use Python 2.7 (  change the Runtime service command to 'python2' in the .exospkg file)
# - update the DEPENDS to python-dev
# find_package(PythonLibs 2)
# c.) use pyenv to manually install a version matching the Python version on the target distro https://realpython.com/intro-to-pyenv/
# set(PYTHON_INCLUDE_PATH ~/.pyenv/versions/3.9-dev/include/python3.9)
# set(PYTHON_LIBRARIES ~/.pyenv/versions/3.9-dev/lib/libpython3.9.so)

include_directories(${PYTHON_INCLUDE_PATH})

include_directories(${CMAKE_CURRENT_SOURCE_DIR})

set(CMAKE_SWIG_FLAGS "")

set(ROS_TOPICS_TYP_SOURCES
    libros_topics_typ.c
    libros_topics_typ.i
    exos_ros_topics_typ.c
    )

set_source_files_properties(${ROS_TOPICS_TYP_SOURCES} PROPERTIES CPLUSPLUS ON)

swig_add_module(libros_topics_typ python ${ROS_TOPICS_TYP_SOURCES})
swig_link_libraries(libros_topics_typ ${PYTHON_LIBRARIES} zmq exos-api)

set(ROS_TOPICS_TYP_MODULE_FILES
    build/_libros_topics_typ.so
    build/libros_topics_typ.py
    )

install(FILES ${ROS_TOPICS_TYP_MODULE_FILES} DESTINATION /home/user/ros_topics_typ)

set(CPACK_GENERATOR "DEB")
set(CPACK_PACKAGE_NAME exos-comp-ros_topics_typ)
set(CPACK_PACKAGE_DESCRIPTION_SUMMARY "ros_topics_typ summary")
set(CPACK_PACKAGE_DESCRIPTION "Some description")
set(CPACK_PACKAGE_VENDOR "Your Company")

set(CPACK_PACKAGE_VERSION_MAJOR 1)
set(CPACK_PACKAGE_VERSION_MINOR 0)
set(CPACK_PACKAGE_VERSION_PATCH 0)
set(CPACK_PACKAGE_FILE_NAME exos-comp-ros_topics_typ_1.0.0_amd64)
set(CPACK_DEBIAN_PACKAGE_MAINTAINER "Your Name")

set(CPACK_DEBIAN_PACKAGE_SHLIBDEPS ON)

include(CPack)
```

- ros_topics_typ.py - Main python script (not shown)

- _libros_topics_typ.so - ros_topics_typ SWIG library (binary file, 581832 bytes)
- ros_topics_typ1.py - Main python script (not shown)

### Program Logical/ros_topics_typ/motorCtrl

#### ros_topics_typ.var
```iecst
VAR
	ros_topics_typInit_0 : ros_topics_typInit;
	ros_topics_typCyclic_0 : ros_topics_typCyclic;
	ros_topics_typExit_0 : ros_topics_typExit;
	ExComponentInfo_0 : ExComponentInfo;
	ExDatamodelInfo_0 : ExDatamodelInfo;
	ros : ros_typ;
	config : REFERENCE TO config_typ;
	hmi : REFERENCE TO hmi_typ;
	hw : REFERENCE TO hw_typ;
	this : REFERENCE TO local_typ;
	localVariables : ARRAY[0..1] OF local_typ;
	watchIdx : USINT;
	k : USINT;
	i : USINT;
END_VAR
```

#### ros_topics_typ.st
```iecst
PROGRAM _INIT

	ros_topics_typInit_0();

	(* Insert code here *)
	FOR i:=0 TO i < 2 BY 1 DO
		setupPointers;

		this.PID.Enable := TRUE;
		this.PID.MinOut := -100;
		this.PID.MaxOut := 100;
		this.PID.PIDParameters.DerivativeTime := 0.00228000456;
		this.PID.PIDParameters.Gain := 78;
		this.PID.PIDParameters.IntegrationTime := 0.02500019;
		this.PID.PIDParameters.FilterTime := 0.000228000456;

		this.PID.Update := TRUE;

		this.PIDCurrent.Enable := TRUE;
		this.PIDCurrent.MinOut := 0;
		this.PIDCurrent.MaxOut := 100;
		this.PIDCurrent.PIDParameters.DerivativeTime := 10;
		this.PIDCurrent.PIDParameters.Gain := 1;
		this.PIDCurrent.PIDParameters.IntegrationTime := 10;
		this.PIDCurrent.PIDParameters.FilterTime := 20;
		this.PIDCurrent.Update := TRUE;
		this.PIDCurrent.SetValue := 8;

		this.filterSpeed.Enable := TRUE;
		this.filterSpeed.WindowLength := 100;
		this.filterSpeed.Update := TRUE;

		this.filterCurrent.Enable := TRUE;
		this.filterCurrent.WindowLength := 3;
		this.filterCurrent.Update := TRUE;

		this.accLimiter.Enable := TRUE;
		this.accLimiter.MaxNegSlewRate := 1;
		this.accLimiter.MaxPosSlewRate := 1;
		this.accLimiter.MaxOut := 2;
		this.accLimiter.MinOut := -2;
		this.accLimiter.Update := TRUE;

		this.PIDtune.SetValue:= 1.0;
		this.PIDtune.MinOut:= 0.0;
		this.PIDtune.MaxOut:= 100.0;
		this.PIDtune.Update := TRUE;

		this.lowPass.Enable := TRUE;
		this.lowPass.CutOffFrequency := 10;
		this.lowPass.Order := 1;
		this.lowPass.Update := TRUE;

		this.encoderOld := this.hw.input.encoder;
		this.timeOld := this.hw.input.nettime;

		this.ton_overcurrent.PT := T#1s;

	END_FOR

END_PROGRAM

PROGRAM _CYCLIC
    //--------------- ex OS ----------------
    //Auto connect:
	ros_topics_typCyclic_0.Enable := ExComponentInfo_0.Operational; // Component has been deployed and started up successfully

	//Auto connect when deployment is off and manually started in GPOS:
	//ros_topics_typCyclic_0.Enable := TRUE;
	ros_topics_typCyclic_0.Start := ros_topics_typCyclic_0.Connected;

	ros_topics_typCyclic_0(Handle := ros_topics_typInit_0.Handle, pros_topics_typ := ADR(ros.topics));

	ExComponentInfo_0(ExTargetLink := ADR(gTarget_0), ExComponentLink := ADR(gros_topics_typ_0), Enable := TRUE);

	ExDatamodelInfo_0(ExTargetLink := ADR(gTarget_0), Enable := TRUE, InstanceName := 'ros_topics_typ_0');
	//--------------- ex OS done ----------------
	ExSyncInfo_0(ExTargetLink := ADR(gTarget_0), Enable := TRUE);

	ros.topics.twist.linear.x := MAX(MIN(ros.topics.twist.linear.x,ros.topics.config.maxSpeed),ros.topics.config.minSpeed);

	IF localVariables[0].hmi.output.overload OR localVariables[1].hmi.output.overload OR NOT ros_topics_typCyclic_0.Operational THEN
		localVariables[0].PID.SetValue := 0;
		localVariables[1].PID.SetValue := 0;
	ELSE
		localVariables[0].PID.SetValue := LREAL_TO_REAL(ros.topics.twist.linear.x + ros.topics.twist.angular.z * ros.topics.config.baseWidth / 2.0) * ros.currentLimiter;  // m/s
		localVariables[1].PID.SetValue := LREAL_TO_REAL(ros.topics.twist.linear.x - ros.topics.twist.angular.z * ros.topics.config.baseWidth / 2.0) * ros.currentLimiter;
	END_IF

	FOR i:=0 TO 1 BY 1 DO
		setupPointers;

		hmi.output.overload := FALSE;

		hmi.output.currentTotal := 0;

		FOR k:=0 TO 7 DO

			hmi.output.current[k] := INT_TO_REAL(hw.input.current[k])*10.0/32767.0;
			hmi.output.currentTotal := hmi.output.currentTotal + hmi.output.current[k];
		END_FOR

		hmi.output.currentTotal := hmi.output.currentTotal /2.0;

		IF this.filterCurrent.UpdateDone THEN
			this.filterSpeed.Update := FALSE;
		END_IF

		this.filterCurrent(In := hmi.output.currentTotal);

		IF this.PIDCurrent.UpdateDone THEN
			this.PIDCurrent.Update := FALSE;
		END_IF

		this.PIDCurrent(ActValue := this.filterCurrent.Out);

		this.currentLimiter := 1;//this.PIDCurrent.Out/100;

		hmi.output.overload := hw.input.overload;

		this.ton_overcurrent(IN := hmi.output.overload);
		IF this.ton_overcurrent.Q THEN
			this.hmi.input.clear := TRUE;
		END_IF

		hw.output.clear := hmi.input.clear;

		IF NOT hmi.output.overload THEN
			hmi.input.clear := FALSE;
		END_IF

		this.diffTime := DINT_TO_LREAL(hw.input.nettime -this.timeOld);
		IF this.diffTime < -100000.0 THEN
			this.diffTime := this.diffTime + 2*2147483647;
		END_IF
		this.diffTime := this.diffTime /1000.0;
		this.timeOld := hw.input.nettime;

		this.diffEncoder := INT_TO_LREAL(hw.input.encoder)-INT_TO_LREAL(this.encoderOld);

		this.encoderOld := hw.input.encoder;

		IF this.diffEncoder > 32727 THEN

			this.diffEncoder := this.diffEncoder - 2*32767;

		ELSIF this.diffEncoder < -32727 THEN

			this.diffEncoder := this.diffEncoder + 2*32767;

		END_IF

		hmi.output.ticks := hmi.output.ticks + this.diffEncoder;
		hmi.output.distance := hmi.output.ticks / UDINT_TO_LREAL(config.ppm);

		IF hmi.input.resetDistance THEN
			hmi.input.resetDistance := FALSE;
			hmi.output.ticks := 0;
			hmi.output.distance := 0;
		END_IF

		this.distance 	:= this.diffEncoder/UDINT_TO_LREAL(config.ppm);

		this.lowPass.In := LREAL_TO_REAL(this.distance);
		this.lowPass();

		this.speed 		:= this.distance * 1000/this.diffTime;

		IF this.filterSpeed.UpdateDone THEN
			this.filterSpeed.Update := FALSE;
		END_IF

		this.filterSpeed(In := LREAL_TO_REAL(this.speed));

		IF this.accLimiter.UpdateDone THEN
			this.accLimiter.Update := FALSE;
		END_IF

		this.accLimiter(In := this.PID.SetValue);

		IF this.PID.UpdateDone THEN
			this.PID.Update := FALSE;
		END_IF

		this.PID.ActValue := LREAL_TO_REAL(this.speed);
		this.PID.SetValue := this.accLimiter.Out;
		// PID TUNE

		IF hmi.input.tune THEN
			this.PIDtune.Enable := TRUE;
		END_IF

		this.PIDtune.ActValue := LREAL_TO_REAL(this.speed);

		IF this.PIDtune.TuningDone THEN
			this.PIDtune.Start := FALSE;
			this.PID.IntegrationPartPresetValue := this.PIDtune.Out;
			this.PID.SetIntegrationPart := TRUE;
		ELSIF this.PIDtune.Active AND NOT this.PIDtune.Update THEN
			//	this.PIDtune.Start := TRUE;
		END_IF

		IF this.PIDtune.UpdateDone THEN
			this.PIDtune.Update := FALSE;
		END_IF

		(* call function block *)
		this.PID();
		this.PIDtune();

		this.PID.SetIntegrationPart := FALSE;

		IF hmi.input.tune THEN
			hw.output.pwm := REAL_TO_INT(this.PIDtune.Out*327.67);
		ELSE
			hw.output.pwm := REAL_TO_INT(this.PID.Out*327.67);
		END_IF

	END_FOR

	ros.currentLimiter := MIN(localVariables[0].currentLimiter,localVariables[1].currentLimiter);

	ros.diffDist := localVariables[1].distance-localVariables[0].distance;
	ros.diffLowpassDist := localVariables[1].lowPass.Out-localVariables[0].lowPass.Out;

	ros.dist := (localVariables[1].distance+localVariables[0].distance)/2;

	IF localVariables[0].diffEncoder = localVariables[1].diffEncoder THEN
		ros.d_theta := 0.0;
		ros.cur_x := ros.cur_x + ros.dist * COS(ros.cur_theta);
		ros.cur_y := ros.cur_y + ros.dist * SIN(ros.cur_theta);
	ELSE
		ros.d_theta := (localVariables[1].distance - localVariables[0].distance) / ros.topics.config.baseWidth;
		ros.dist := (localVariables[1].distance+localVariables[0].distance)/2;
		ros.r := ros.dist / ros.d_theta;
		ros.cur_x := ros.cur_x + ros.r * (SIN(ros.d_theta + ros.cur_theta) - SIN(ros.cur_theta));
		ros.cur_y := ros.cur_y - ros.r * (COS(ros.d_theta + ros.cur_theta) - COS(ros.cur_theta));
		ros.cur_theta := normalizeAngle(ros.cur_theta + ros.d_theta);
	END_IF

	ros.vel_x := ros.dist * (1000.0/localVariables[0].diffTime);
	ros.vel_theta := ros.d_theta * (1000.0/localVariables[0].diffTime);

	// set ros data
	ros.topics.odemetry.pose.pose.position.x 	:= ros.cur_x;
	ros.topics.odemetry.pose.pose.position.y	:= ros.cur_y;
	ros.topics.odemetry.pose.pose.orientation.z	:= ros.cur_theta;

	ros.topics.odemetry.twist.twist.linear.x  	:= ros.vel_x;
	ros.topics.odemetry.twist.twist.angular.z 	:= ros.vel_theta;

	setupWatchPointers;

END_PROGRAM

PROGRAM _EXIT

	ros_topics_typExit_0(Handle := ros_topics_typInit_0.Handle);

END_PROGRAM
```

#### setupPointers.st
```iecst
ACTION setupPointers:

	this ACCESS ADR(localVariables[i]);
	config ACCESS ADR(localVariables[i].hmi.config);
	hw ACCESS ADR(localVariables[i].hw);
	hmi ACCESS ADR(localVariables[i].hmi);

END_ACTION

ACTION setupWatchPointers:

	i := watchIdx;
	this ACCESS ADR(localVariables[i]);
	config ACCESS ADR(localVariables[i].hmi.config);
	hw ACCESS ADR(localVariables[i].hw);
	hmi ACCESS ADR(localVariables[i].hmi);

END_ACTION
```

### ros_topics_typ.var
```iecst
VAR
    ros_topics_typInit_0 : ros_topics_typInit;
    ros_topics_typCyclic_0 : ros_topics_typCyclic;
    ros_topics_typExit_0 : ros_topics_typExit;
    ros_topics_typ_0 : ros_topics_typ;
    ExComponentInfo_0 : ExComponentInfo;
    ExDatamodelInfo_0 : ExDatamodelInfo;
END_VAR
```

### Program Logical/ros_topics_typ - Copy/motorCtrl (IEC) - ros_topics_typ application

#### motorCtrl.typ - Local data types
```iecst
TYPE
	ros_typ : 	STRUCT
		vel_theta : LREAL;
		vel_x : LREAL;
		r : LREAL;
		cur_theta : LREAL;
		dist : LREAL;
		cur_y : LREAL;
		cur_x : LREAL;
		d_theta : LREAL;
		topics : ros_topics_typ;
		diffLowpassDist : REAL;
		diffDist : LREAL;
		currentLimiter : REAL;
	END_STRUCT;
	local_typ : 	STRUCT
		hw : hw_typ;
		hmi : hmi_typ;
		speed : LREAL;
		encoderOld : INT;
		accLimiter : MTBasicsLimiter;
		PIDCurrent : MTBasicsPID;
		PID : MTBasicsPID;
		distance : LREAL;
		diffEncoder : LREAL;
		filterCurrent : MTFilterMovingAverage;
		filterSpeed : MTFilterMovingAverage;
		diffTime : LREAL;
		timeOld : DINT;
		PIDtune : MTBasicsOscillationTuning;
		lowPass : MTFilterLowPass;
		ton_overcurrent : TON;
		currentLimiter : REAL;
	END_STRUCT;
	hw_typ : 	STRUCT
		input : hw_input_typ;
		output : hw_output_typ;
	END_STRUCT;
	hw_output_typ : 	STRUCT
		pwm : INT;
		clear : BOOL;
	END_STRUCT;
	hw_input_typ : 	STRUCT
		encoder : INT;
		overload : BOOL;
		current : ARRAY[0..7]OF INT;
		nettime : DINT;
	END_STRUCT;
	hmi_typ : 	STRUCT
		config : config_typ;
		output : hmi_output_typ;
		input : hmi_input_typ;
	END_STRUCT;
	hmi_output_typ : 	STRUCT
		current : ARRAY[0..7]OF REAL;
		overload : BOOL;
		distance : LREAL;
		ticks : LREAL;
		currentTotal : REAL;
	END_STRUCT;
	hmi_input_typ : 	STRUCT
		clear : BOOL;
		tune : BOOL;
		resetDistance : BOOL;
	END_STRUCT;
	config_typ : 	STRUCT
		ppm : UDINT := 105860;
		maxCurrent : REAL := 8;
	END_STRUCT;
	common_typ : 	STRUCT
	END_STRUCT;
END_TYPE
```

#### ros_topics_typ.var - ros_topics_typ variable declaration
```iecst
VAR
	ros_topics_typInit_0 : ros_topics_typInit;
	ros_topics_typCyclic_0 : ros_topics_typCyclic;
	ros_topics_typExit_0 : ros_topics_typExit;
	ExComponentInfo_0 : ExComponentInfo;
	ExSyncInfo_0 : ExSyncInfo;
	ExDatamodelInfo_0 : ExDatamodelInfo;
	ros : ros_typ;
	config : REFERENCE TO config_typ;
	hmi : REFERENCE TO hmi_typ;
	hw : REFERENCE TO hw_typ;
	this : REFERENCE TO local_typ;
	localVariables : ARRAY[0..1] OF local_typ;
	watchIdx : USINT;
	k : USINT;
	i : USINT;
END_VAR
```

### Library Logical/ros_topics_typ - Copy/ros_topics (ANSIC) - ros_topics_typ exOS library
Depends on: ExData

#### exos_ros_topics_typ.c - Generated datamodel source for ros_topics_typ
```c
/*Automatically generated c file from ros_topics_typ.typ*/

#include "exos_ros_topics_typ.h"

const char config_ros_topics_typ[] = "{\"name\":\"struct\",\"attributes\":{\"name\":\"<NAME>\",\"dataType\":\"ros_topics_typ\",\"info\":\"<infoId0>\"},\"children\":[{\"name\":\"struct\",\"attributes\":{\"name\":\"odemetry\",\"dataType\":\"ros_topic_odemety_typ\",\"comment\":\"PUB\",\"info\":\"<infoId1>\"},\"children\":[{\"name\":\"struct\",\"attributes\":{\"name\":\"pose\",\"dataType\":\"ros_topic_poseCor_typ\",\"info\":\"<infoId2>\"},\"children\":[{\"name\":\"struct\",\"attributes\":{\"name\":\"pose\",\"dataType\":\"ros_topic_pose_typ\",\"info\":\"<infoId3>\"},\"children\":[{\"name\":\"struct\",\"attributes\":{\"name\":\"position\",\"dataType\":\"ros_topic_point_typ\",\"info\":\"<infoId4>\"},\"children\":[{\"name\":\"variable\",\"attributes\":{\"name\":\"y\",\"dataType\":\"LREAL\",\"info\":\"<infoId5>\"}},{\"name\":\"variable\",\"attributes\":{\"name\":\"z\",\"dataType\":\"LREAL\",\"info\":\"<infoId6>\"}},{\"name\":\"variable\",\"attributes\":{\"name\":\"x\",\"dataType\":\"LREAL\",\"info\":\"<infoId7>\"}}]},{\"name\":\"struct\",\"attributes\":{\"name\":\"orientation\",\"dataType\":\"ros_topic_quaternion_typ\",\"info\":\"<infoId8>\"},\"children\":[{\"name\":\"variable\",\"attributes\":{\"name\":\"y\",\"dataType\":\"LREAL\",\"info\":\"<infoId9>\"}},{\"name\":\"variable\",\"attributes\":{\"name\":\"z\",\"dataType\":\"LREAL\",\"info\":\"<infoId10>\"}},{\"name\":\"variable\",\"attributes\":{\"name\":\"w\",\"dataType\":\"LREAL\",\"info\":\"<infoId11>\"}},{\"name\":\"variable\",\"attributes\":{\"name\":\"x\",\"dataType\":\"LREAL\",\"info\":\"<infoId12>\"}}]}]}]},{\"name\":\"struct\",\"attributes\":{\"name\":\"twist\",\"dataType\":\"ros_topic_twistCor_typ\",\"info\":\"<infoId13>\"},\"children\":[{\"name\":\"struct\",\"attributes\":{\"name\":\"twist\",\"dataType\":\"ros_topic_twist_typ\",\"info\":\"<infoId14>\"},\"children\":[{\"name\":\"struct\",\"attributes\":{\"name\":\"angular\",\"dataType\":\"ros_topic_vector3_typ\",\"info\":\"<infoId15>\"},\"children\":[{\"name\":\"variable\",\"attributes\":{\"name\":\"y\",\"dataType\":\"LREAL\",\"info\":\"<infoId16>\"}},{\"name\":\"variable\",\"attributes\":{\"name\":\"z\",\"dataType\":\"LREAL\",\"info\":\"<infoId17>\"}},{\"name\":\"variable\",\"attributes\":{\"name\":\"x\",\"dataType\":\"LREAL\",\"info\":\"<infoId18>\"}}]},{\"name\":\"struct\",\"attributes\":{\"name\":\"linear\",\"dataType\":\"ros_topic_vector3_typ\",\"info\":\"<infoId19>\"},\"children\":[{\"name\":\"variable\",\"attributes\":{\"name\":\"y\",\"dataType\":\"LREAL\",\"info\":\"<infoId20>\"}},{\"name\":\"variable\",\"attributes\":{\"name\":\"z\",\"dataType\":\"LREAL\",\"info\":\"<infoId21>\"}},{\"name\":\"variable\",\"attributes\":{\"name\":\"x\",\"dataType\":\"LREAL\",\"info\":\"<infoId22>\"}}]}]}]},{\"name\":\"struct\",\"attributes\":{\"name\":\"header\",\"dataType\":\"ros_topic_header_typ\",\"info\":\"<infoId23>\"},\"children\":[{\"name\":\"struct\",\"attributes\":{\"name\":\"stamp\",\"dataType\":\"ros_topic_time_typ\",\"info\":\"<infoId24>\"},\"children\":[{\"name\":\"variable\",\"attributes\":{\"name\":\"nsec\",\"dataType\":\"UDINT\",\"info\":\"<infoId25>\"}},{\"name\":\"variable\",\"attributes\":{\"name\":\"sec\",\"dataType\":\"UDINT\",\"info\":\"<infoId26>\"}}]},{\"name\":\"variable\",\"attributes\":{\"name\":\"seq\",\"dataType\":\"UDINT\",\"info\":\"<infoId27>\"}},{\"name\":\"variable\",\"attributes\":{\"name\":\"frame_id\",\"dataType\":\"STRING\",\"stringLength\":21,\"info\":\"<infoId28>\"}}]}]},{\"name\":\"struct\",\"attributes\":{\"name\":\"twist\",\"dataType\":\"ros_topic_twist_typ\",\"comment\":\"SUB\",\"info\":\"<infoId29>\"},\"children\":[{\"name\":\"struct\",\"attributes\":{\"name\":\"angular\",\"dataType\":\"ros_topic_vector3_typ\",\"info\":\"<infoId30>\"},\"children\":[{\"name\":\"variable\",\"attributes\":{\"name\":\"y\",\"dataType\":\"LREAL\",\"info\":\"<infoId31>\"}},{\"name\":\"variable\",\"attributes\":{\"name\":\"z\",\"dataType\":\"LREAL\",\"info\":\"<infoId32>\"}},{\"name\":\"variable\",\"attributes\":{\"name\":\"x\",\"dataType\":\"LREAL\",\"info\":\"<infoId33>\"}}]},{\"name\":\"struct\",\"attributes\":{\"name\":\"linear\",\"dataType\":\"ros_topic_vector3_typ\",\"info\":\"<infoId34>\"},\"children\":[{\"name\":\"variable\",\"attributes\":{\"name\":\"y\",\"dataType\":\"LREAL\",\"info\":\"<infoId35>\"}},{\"name\":\"variable\",\"attributes\":{\"name\":\"z\",\"dataType\":\"LREAL\",\"info\":\"<infoId36>\"}},{\"name\":\"variable\",\"attributes\":{\"name\":\"x\",\"dataType\":\"LREAL\",\"info\":\"<infoId37>\"}}]}]},{\"name\":\"struct\",\"attributes\":{\"name\":\"config\",\"dataType\":\"ros_config_typ\",\"comment\":\"SUB\",\"info\":\"<infoId38>\"},\"children\":[{\"name\":\"variable\",\"attributes\":{\"name\":\"maxSpeed\",\"dataType\":\"LREAL\",\"info\":\"<infoId39>\"}},{\"name\":\"variable\",\"attributes\":{\"name\":\"minSpeed\",\"dataType\":\"LREAL\",\"info\":\"<infoId40>\"}},{\"name\":\"variable\",\"attributes\":{\"name\":\"baseWidth\",\"dataType\":\"LREAL\",\"info\":\"<infoId41>\"}}]}]}";

/*Connect the ros_topics_typ datamodel to the server*/
EXOS_ERROR_CODE exos_datamodel_connect_ros_topics_typ(exos_datamodel_handle_t *datamodel, exos_datamodel_event_cb datamodel_event_callback)
{
    ros_topics_typ data;
    exos_dataset_info_t datasets[] = {
        {EXOS_DATASET_BROWSE_NAME_INIT,{}},
        {EXOS_DATASET_BROWSE_NAME(odemetry),{}},
        {EXOS_DATASET_BROWSE_NAME(odemetry.pose),{}},
        {EXOS_DATASET_BROWSE_NAME(odemetry.pose.pose),{}},
        {EXOS_DATASET_BROWSE_NAME(odemetry.pose.pose.position),{}},
        {EXOS_DATASET_BROWSE_NAME(odemetry.pose.pose.position.y),{}},
        {EXOS_DATASET_BROWSE_NAME(odemetry.pose.pose.position.z),{}},
        {EXOS_DATASET_BROWSE_NAME(odemetry.pose.pose.position.x),{}},
        {EXOS_DATASET_BROWSE_NAME(odemetry.pose.pose.orientation),{}},
        {EXOS_DATASET_BROWSE_NAME(odemetry.pose.pose.orientation.y),{}},
        {EXOS_DATASET_BROWSE_NAME(odemetry.pose.pose.orientation.z),{}},
        {EXOS_DATASET_BROWSE_NAME(odemetry.pose.pose.orientation.w),{}},
        {EXOS_DATASET_BROWSE_NAME(odemetry.pose.pose.orientation.x),{}},
        {EXOS_DATASET_BROWSE_NAME(odemetry.twist),{}},
        {EXOS_DATASET_BROWSE_NAME(odemetry.twist.twist),{}},
        {EXOS_DATASET_BROWSE_NAME(odemetry.twist.twist.angular),{}},
        {EXOS_DATASET_BROWSE_NAME(odemetry.twist.twist.angular.y),{}},
        {EXOS_DATASET_BROWSE_NAME(odemetry.twist.twist.angular.z),{}},
        {EXOS_DATASET_BROWSE_NAME(odemetry.twist.twist.angular.x),{}},
        {EXOS_DATASET_BROWSE_NAME(odemetry.twist.twist.linear),{}},
        {EXOS_DATASET_BROWSE_NAME(odemetry.twist.twist.linear.y),{}},
        {EXOS_DATASET_BROWSE_NAME(odemetry.twist.twist.linear.z),{}},
        {EXOS_DATASET_BROWSE_NAME(odemetry.twist.twist.linear.x),{}},
        {EXOS_DATASET_BROWSE_NAME(odemetry.header),{}},
        {EXOS_DATASET_BROWSE_NAME(odemetry.header.stamp),{}},
        {EXOS_DATASET_BROWSE_NAME(odemetry.header.stamp.nsec),{}},
        {EXOS_DATASET_BROWSE_NAME(odemetry.header.stamp.sec),{}},
        {EXOS_DATASET_BROWSE_NAME(odemetry.header.seq),{}},
        {EXOS_DATASET_BROWSE_NAME(odemetry.header.frame_id),{}},
        {EXOS_DATASET_BROWSE_NAME(twist),{}},
        {EXOS_DATASET_BROWSE_NAME(twist.angular),{}},
        {EXOS_DATASET_BROWSE_NAME(twist.angular.y),{}},
        {EXOS_DATASET_BROWSE_NAME(twist.angular.z),{}},
        {EXOS_DATASET_BROWSE_NAME(twist.angular.x),{}},
        {EXOS_DATASET_BROWSE_NAME(twist.linear),{}},
        {EXOS_DATASET_BROWSE_NAME(twist.linear.y),{}},
        {EXOS_DATASET_BROWSE_NAME(twist.linear.z),{}},
        {EXOS_DATASET_BROWSE_NAME(twist.linear.x),{}},
        {EXOS_DATASET_BROWSE_NAME(config),{}},
        {EXOS_DATASET_BROWSE_NAME(config.maxSpeed),{}},
        {EXOS_DATASET_BROWSE_NAME(config.minSpeed),{}},
        {EXOS_DATASET_BROWSE_NAME(config.baseWidth),{}}
    };

    exos_datamodel_calc_dataset_info(datasets, sizeof(datasets));

    return exos_datamodel_connect(datamodel, config_ros_topics_typ, datasets, sizeof(datasets), datamodel_event_callback);
}
```

### Package Logical/ros_topics_typ - Copy/Linux - ros_topics_typ Linux resources

### exos_ros_topics_typ.h
```c
/*Automatically generated header file from ros_topics_typ.typ*/

#ifndef _EXOS_COMP_ROS_TOPICS_TYP_H_
#define _EXOS_COMP_ROS_TOPICS_TYP_H_

#include "exos_api.h"

#if defined(_SG4)
#include <ros_topics.h>
#else
#include <stddef.h>
#include <stdint.h>
#include <stdbool.h>

typedef struct ros_config_typ
{
    double maxSpeed;
    double minSpeed;
    double baseWidth;

} ros_config_typ;

typedef struct ros_topic_vector3_typ
{
    double y;
    double z;
    double x;

} ros_topic_vector3_typ;

typedef struct ros_topic_twist_typ
{
    struct ros_topic_vector3_typ angular;
    struct ros_topic_vector3_typ linear;

} ros_topic_twist_typ;

typedef struct ros_topic_time_typ
{
    uint32_t nsec;
    uint32_t sec;

} ros_topic_time_typ;

typedef struct ros_topic_header_typ
{
    struct ros_topic_time_typ stamp;
    uint32_t seq;
    char frame_id[21];

} ros_topic_header_typ;

typedef struct ros_topic_twistCor_typ
{
    struct ros_topic_twist_typ twist;

} ros_topic_twistCor_typ;

typedef struct ros_topic_quaternion_typ
{
    double y;
    double z;
    double w;
    double x;

} ros_topic_quaternion_typ;

typedef struct ros_topic_point_typ
{
    double y;
    double z;
    double x;

} ros_topic_point_typ;

typedef struct ros_topic_pose_typ
{
    struct ros_topic_point_typ position;
    struct ros_topic_quaternion_typ orientation;

} ros_topic_pose_typ;

typedef struct ros_topic_poseCor_typ
{
    struct ros_topic_pose_typ pose;

} ros_topic_poseCor_typ;

typedef struct ros_topic_odemety_typ
{
    struct ros_topic_poseCor_typ pose;
    struct ros_topic_twistCor_typ twist;
    struct ros_topic_header_typ header;

} ros_topic_odemety_typ;

typedef struct ros_topics_typ
{
    struct ros_topic_odemety_typ odemetry; //PUB
    struct ros_topic_twist_typ twist; //SUB
    struct ros_config_typ config; //SUB

} ros_topics_typ;

#endif // _SG4

EXOS_ERROR_CODE exos_datamodel_connect_ros_topics_typ(exos_datamodel_handle_t *datamodel, exos_datamodel_event_cb datamodel_event_callback);

#endif // _EXOS_COMP_ROS_TOPICS_TYP_H_
```

- libros_topics_typ.py (not shown)

- ros_topics_typ.py (not shown)

### ros_topics.typ
```iecst
TYPE
	ros_topic_point_typ : 	STRUCT  (*this expresses velocity in free space broken into its linear and angular parts.*)
		y : LREAL;
		z : LREAL;
		x : LREAL;
	END_STRUCT;
	ros_topic_vector3_typ : 	STRUCT  (*this expresses velocity in free space broken into its linear and angular parts.*)
		y : LREAL;
		z : LREAL;
		x : LREAL;
	END_STRUCT;
	ros_topic_twist_typ : 	STRUCT  (*This expresses velocity in free space broken into its linear and angular parts.*)
		angular : ros_topic_vector3_typ;
		linear : ros_topic_vector3_typ;
	END_STRUCT;
	ros_topic_twistCor_typ : 	STRUCT  (*This expresses velocity in free space with uncertainty.*)
		twist : ros_topic_twist_typ;
	END_STRUCT;
	ros_topic_quaternion_typ : 	STRUCT  (*This represents an orientation in free space in quaternion form.*)
		y : LREAL;
		z : LREAL;
		w : LREAL;
		x : LREAL;
	END_STRUCT;
	ros_topic_odemety_point_typ : 	STRUCT  (*This contains the position of a point in free space*)
		y : LREAL;
		z : LREAL;
		x : LREAL;
	END_STRUCT;
	ros_topic_pose_typ : 	STRUCT  (*A representation of pose in free space, composed of position and orientation. *)
		position : ros_topic_point_typ;
		orientation : ros_topic_quaternion_typ;
	END_STRUCT;
	ros_topic_poseCor_typ : 	STRUCT  (*This represents a pose in free space with uncertainty.*)
		pose : ros_topic_pose_typ;
	END_STRUCT;
	ros_topic_time_typ : 	STRUCT
		nsec : UDINT;
		sec : UDINT;
	END_STRUCT;
	ros_topic_header_typ : 	STRUCT
		stamp : ros_topic_time_typ;
		seq : UDINT;
		frame_id : STRING[20];
	END_STRUCT;
	ros_topic_odemety_typ : 	STRUCT
		pose : ros_topic_poseCor_typ;
		twist : ros_topic_twistCor_typ;
		header : ros_topic_header_typ;
	END_STRUCT;
	ros_config_typ : 	STRUCT
		maxSpeed : LREAL := 2;
		minSpeed : LREAL := -2;
		baseWidth : LREAL := 0.53;
	END_STRUCT;
	ros_topics_typ : 	STRUCT
		odemetry : ros_topic_odemety_typ; (*PUB*)
		twist : ros_topic_twist_typ; (*SUB*)
		config : ros_config_typ; (*SUB*)
	END_STRUCT;
	ros_motorCtrl : 	STRUCT
		twist : ros_topic_twist_typ; (*SUB*)
		config : ros_config_typ; (*SUB*)
	END_STRUCT;
END_TYPE
```

### Program Logical/test/ros_topics_typ/ros_topics_0 (IEC) - ros_topics_typ application

#### ros_topics_typ.st - ros_topics_typ application
```iecst
PROGRAM _INIT

    ros_topics_typInit_0();

END_PROGRAM

PROGRAM _CYCLIC

    //Auto connect:
    //ros_topics_typCyclic_0.Enable := ExComponentInfo_0.Operational; // Component has been deployed and started up successfully

    ros_topics_typCyclic_0(Handle := ros_topics_typInit_0.Handle, pros_topics_typ := ADR(ros_topics_typ_0));

    ExComponentInfo_0(ExTargetLink := ADR(gTarget_0), ExComponentLink := ADR(gros_topics_typ_0), Enable := TRUE);

    ExDatamodelInfo_0(ExTargetLink := ADR(gTarget_0), Enable := TRUE, InstanceName := 'ros_topics_typ_0');

END_PROGRAM

PROGRAM _EXIT

    ros_topics_typExit_0(Handle := ros_topics_typInit_0.Handle);

END_PROGRAM
```

### Library Logical/test/ros_topics_typ/ros_topics (ANSIC) - ros_topics_typ exOS library

#### exos_ros_topics_typ.c
```c
/*Automatically generated c file from ros_topics.typ*/

#include "exos_ros_topics_typ.h"

const char config_ros_topics_typ[] = "{\"name\":\"struct\",\"attributes\":{\"name\":\"<NAME>\",\"dataType\":\"ros_topics_typ\",\"info\":\"<infoId0>\"},\"children\":[{\"name\":\"struct\",\"attributes\":{\"name\":\"odemetry\",\"dataType\":\"ros_topic_odemety_typ\",\"comment\":\"PUB\",\"info\":\"<infoId1>\"},\"children\":[{\"name\":\"struct\",\"attributes\":{\"name\":\"pose\",\"dataType\":\"ros_topic_poseCor_typ\",\"info\":\"<infoId2>\"},\"children\":[{\"name\":\"struct\",\"attributes\":{\"name\":\"pose\",\"dataType\":\"ros_topic_pose_typ\",\"info\":\"<infoId3>\"},\"children\":[{\"name\":\"struct\",\"attributes\":{\"name\":\"position\",\"dataType\":\"ros_topic_point_typ\",\"info\":\"<infoId4>\"},\"children\":[{\"name\":\"variable\",\"attributes\":{\"name\":\"y\",\"dataType\":\"LREAL\",\"info\":\"<infoId5>\"}},{\"name\":\"variable\",\"attributes\":{\"name\":\"z\",\"dataType\":\"LREAL\",\"info\":\"<infoId6>\"}},{\"name\":\"variable\",\"attributes\":{\"name\":\"x\",\"dataType\":\"LREAL\",\"info\":\"<infoId7>\"}}]},{\"name\":\"struct\",\"attributes\":{\"name\":\"orientation\",\"dataType\":\"ros_topic_quaternion_typ\",\"info\":\"<infoId8>\"},\"children\":[{\"name\":\"variable\",\"attributes\":{\"name\":\"y\",\"dataType\":\"LREAL\",\"info\":\"<infoId9>\"}},{\"name\":\"variable\",\"attributes\":{\"name\":\"z\",\"dataType\":\"LREAL\",\"info\":\"<infoId10>\"}},{\"name\":\"variable\",\"attributes\":{\"name\":\"w\",\"dataType\":\"LREAL\",\"info\":\"<infoId11>\"}},{\"name\":\"variable\",\"attributes\":{\"name\":\"x\",\"dataType\":\"LREAL\",\"info\":\"<infoId12>\"}}]}]}]},{\"name\":\"struct\",\"attributes\":{\"name\":\"twist\",\"dataType\":\"ros_topic_twistCor_typ\",\"info\":\"<infoId13>\"},\"children\":[{\"name\":\"struct\",\"attributes\":{\"name\":\"twist\",\"dataType\":\"ros_topic_twist_typ\",\"info\":\"<infoId14>\"},\"children\":[{\"name\":\"struct\",\"attributes\":{\"name\":\"angular\",\"dataType\":\"ros_topic_vector3_typ\",\"info\":\"<infoId15>\"},\"children\":[{\"name\":\"variable\",\"attributes\":{\"name\":\"y\",\"dataType\":\"LREAL\",\"info\":\"<infoId16>\"}},{\"name\":\"variable\",\"attributes\":{\"name\":\"z\",\"dataType\":\"LREAL\",\"info\":\"<infoId17>\"}},{\"name\":\"variable\",\"attributes\":{\"name\":\"x\",\"dataType\":\"LREAL\",\"info\":\"<infoId18>\"}}]},{\"name\":\"struct\",\"attributes\":{\"name\":\"linear\",\"dataType\":\"ros_topic_vector3_typ\",\"info\":\"<infoId19>\"},\"children\":[{\"name\":\"variable\",\"attributes\":{\"name\":\"y\",\"dataType\":\"LREAL\",\"info\":\"<infoId20>\"}},{\"name\":\"variable\",\"attributes\":{\"name\":\"z\",\"dataType\":\"LREAL\",\"info\":\"<infoId21>\"}},{\"name\":\"variable\",\"attributes\":{\"name\":\"x\",\"dataType\":\"LREAL\",\"info\":\"<infoId22>\"}}]}]}]},{\"name\":\"struct\",\"attributes\":{\"name\":\"header\",\"dataType\":\"ros_topic_header_typ\",\"info\":\"<infoId23>\"},\"children\":[{\"name\":\"struct\",\"attributes\":{\"name\":\"stamp\",\"dataType\":\"ros_topic_time_typ\",\"info\":\"<infoId24>\"},\"children\":[{\"name\":\"variable\",\"attributes\":{\"name\":\"nsec\",\"dataType\":\"UDINT\",\"info\":\"<infoId25>\"}},{\"name\":\"variable\",\"attributes\":{\"name\":\"sec\",\"dataType\":\"UDINT\",\"info\":\"<infoId26>\"}}]},{\"name\":\"variable\",\"attributes\":{\"name\":\"seq\",\"dataType\":\"UDINT\",\"info\":\"<infoId27>\"}},{\"name\":\"variable\",\"attributes\":{\"name\":\"frame_id\",\"dataType\":\"STRING\",\"stringLength\":21,\"info\":\"<infoId28>\"}}]}]},{\"name\":\"struct\",\"attributes\":{\"name\":\"twist\",\"dataType\":\"ros_topic_twist_typ\",\"comment\":\"SUB\",\"info\":\"<infoId29>\"},\"children\":[{\"name\":\"struct\",\"attributes\":{\"name\":\"angular\",\"dataType\":\"ros_topic_vector3_typ\",\"info\":\"<infoId30>\"},\"children\":[{\"name\":\"variable\",\"attributes\":{\"name\":\"y\",\"dataType\":\"LREAL\",\"info\":\"<infoId31>\"}},{\"name\":\"variable\",\"attributes\":{\"name\":\"z\",\"dataType\":\"LREAL\",\"info\":\"<infoId32>\"}},{\"name\":\"variable\",\"attributes\":{\"name\":\"x\",\"dataType\":\"LREAL\",\"info\":\"<infoId33>\"}}]},{\"name\":\"struct\",\"attributes\":{\"name\":\"linear\",\"dataType\":\"ros_topic_vector3_typ\",\"info\":\"<infoId34>\"},\"children\":[{\"name\":\"variable\",\"attributes\":{\"name\":\"y\",\"dataType\":\"LREAL\",\"info\":\"<infoId35>\"}},{\"name\":\"variable\",\"attributes\":{\"name\":\"z\",\"dataType\":\"LREAL\",\"info\":\"<infoId36>\"}},{\"name\":\"variable\",\"attributes\":{\"name\":\"x\",\"dataType\":\"LREAL\",\"info\":\"<infoId37>\"}}]}]},{\"name\":\"struct\",\"attributes\":{\"name\":\"config\",\"dataType\":\"ros_config_typ\",\"comment\":\"SUB\",\"info\":\"<infoId38>\"},\"children\":[{\"name\":\"variable\",\"attributes\":{\"name\":\"maxSpeed\",\"dataType\":\"LREAL\",\"info\":\"<infoId39>\"}},{\"name\":\"variable\",\"attributes\":{\"name\":\"minSpeed\",\"dataType\":\"LREAL\",\"info\":\"<infoId40>\"}},{\"name\":\"variable\",\"attributes\":{\"name\":\"baseWidth\",\"dataType\":\"LREAL\",\"info\":\"<infoId41>\"}}]}]}";

/*Connect the ros_topics_typ datamodel to the server*/
EXOS_ERROR_CODE exos_datamodel_connect_ros_topics_typ(exos_datamodel_handle_t *datamodel, exos_datamodel_event_cb datamodel_event_callback)
{
    ros_topics_typ data;
    exos_dataset_info_t datasets[] = {
        {EXOS_DATASET_BROWSE_NAME_INIT,{}},
        {EXOS_DATASET_BROWSE_NAME(odemetry),{}},
        {EXOS_DATASET_BROWSE_NAME(odemetry.pose),{}},
        {EXOS_DATASET_BROWSE_NAME(odemetry.pose.pose),{}},
        {EXOS_DATASET_BROWSE_NAME(odemetry.pose.pose.position),{}},
        {EXOS_DATASET_BROWSE_NAME(odemetry.pose.pose.position.y),{}},
        {EXOS_DATASET_BROWSE_NAME(odemetry.pose.pose.position.z),{}},
        {EXOS_DATASET_BROWSE_NAME(odemetry.pose.pose.position.x),{}},
        {EXOS_DATASET_BROWSE_NAME(odemetry.pose.pose.orientation),{}},
        {EXOS_DATASET_BROWSE_NAME(odemetry.pose.pose.orientation.y),{}},
        {EXOS_DATASET_BROWSE_NAME(odemetry.pose.pose.orientation.z),{}},
        {EXOS_DATASET_BROWSE_NAME(odemetry.pose.pose.orientation.w),{}},
        {EXOS_DATASET_BROWSE_NAME(odemetry.pose.pose.orientation.x),{}},
        {EXOS_DATASET_BROWSE_NAME(odemetry.twist),{}},
        {EXOS_DATASET_BROWSE_NAME(odemetry.twist.twist),{}},
        {EXOS_DATASET_BROWSE_NAME(odemetry.twist.twist.angular),{}},
        {EXOS_DATASET_BROWSE_NAME(odemetry.twist.twist.angular.y),{}},
        {EXOS_DATASET_BROWSE_NAME(odemetry.twist.twist.angular.z),{}},
        {EXOS_DATASET_BROWSE_NAME(odemetry.twist.twist.angular.x),{}},
        {EXOS_DATASET_BROWSE_NAME(odemetry.twist.twist.linear),{}},
        {EXOS_DATASET_BROWSE_NAME(odemetry.twist.twist.linear.y),{}},
        {EXOS_DATASET_BROWSE_NAME(odemetry.twist.twist.linear.z),{}},
        {EXOS_DATASET_BROWSE_NAME(odemetry.twist.twist.linear.x),{}},
        {EXOS_DATASET_BROWSE_NAME(odemetry.header),{}},
        {EXOS_DATASET_BROWSE_NAME(odemetry.header.stamp),{}},
        {EXOS_DATASET_BROWSE_NAME(odemetry.header.stamp.nsec),{}},
        {EXOS_DATASET_BROWSE_NAME(odemetry.header.stamp.sec),{}},
        {EXOS_DATASET_BROWSE_NAME(odemetry.header.seq),{}},
        {EXOS_DATASET_BROWSE_NAME(odemetry.header.frame_id),{}},
        {EXOS_DATASET_BROWSE_NAME(twist),{}},
        {EXOS_DATASET_BROWSE_NAME(twist.angular),{}},
        {EXOS_DATASET_BROWSE_NAME(twist.angular.y),{}},
        {EXOS_DATASET_BROWSE_NAME(twist.angular.z),{}},
        {EXOS_DATASET_BROWSE_NAME(twist.angular.x),{}},
        {EXOS_DATASET_BROWSE_NAME(twist.linear),{}},
        {EXOS_DATASET_BROWSE_NAME(twist.linear.y),{}},
        {EXOS_DATASET_BROWSE_NAME(twist.linear.z),{}},
        {EXOS_DATASET_BROWSE_NAME(twist.linear.x),{}},
        {EXOS_DATASET_BROWSE_NAME(config),{}},
        {EXOS_DATASET_BROWSE_NAME(config.maxSpeed),{}},
        {EXOS_DATASET_BROWSE_NAME(config.minSpeed),{}},
        {EXOS_DATASET_BROWSE_NAME(config.baseWidth),{}}
    };

    exos_datamodel_calc_dataset_info(datasets, sizeof(datasets));

    return exos_datamodel_connect(datamodel, config_ros_topics_typ, datasets, sizeof(datasets), datamodel_event_callback);
}
```

#### ros_topics_typ.c
```c
#include <ros_topics.h>

#define EXOS_ASSERT_LOG &handle->logger
#define EXOS_ASSERT_CALLBACK inst->_state = 255;
#include "exos_log.h"
#include "exos_ros_topics_typ.h"
#include <string.h>

#define SUCCESS(_format_, ...) exos_log_success(&handle->logger, EXOS_LOG_TYPE_USER, _format_, ##__VA_ARGS__);
#define INFO(_format_, ...) exos_log_info(&handle->logger, EXOS_LOG_TYPE_USER, _format_, ##__VA_ARGS__);
#define VERBOSE(_format_, ...) exos_log_debug(&handle->logger, EXOS_LOG_TYPE_USER + EXOS_LOG_TYPE_VERBOSE, _format_, ##__VA_ARGS__);
#define ERROR(_format_, ...) exos_log_error(&handle->logger, _format_, ##__VA_ARGS__);

typedef struct
{
    void *self;
    exos_log_handle_t logger;
    ros_topics_typ data;

    exos_datamodel_handle_t ros_topics_typ_datamodel;

    exos_dataset_handle_t odemetry_dataset;
    exos_dataset_handle_t twist_dataset;
    exos_dataset_handle_t config_dataset;
} ros_topics_typHandle_t;

static void datasetEvent(exos_dataset_handle_t *dataset, EXOS_DATASET_EVENT_TYPE event_type, void *info)
{
    struct ros_topics_typCyclic *inst = (struct ros_topics_typCyclic *)dataset->datamodel->user_context;
    ros_topics_typHandle_t *handle = (ros_topics_typHandle_t *)inst->Handle;

    switch (event_type)
    {
    case EXOS_DATASET_EVENT_UPDATED:
        VERBOSE("dataset %s updated! latency (us):%i", dataset->name, (exos_datamodel_get_nettime(dataset->datamodel) - dataset->nettime));
        //handle each subscription dataset separately
        if(0 == strcmp(dataset->name, "twist"))
        {
            memcpy(&inst->pros_topics_typ->twist, dataset->data, dataset->size);
        }
        else if(0 == strcmp(dataset->name, "config"))
        {
            memcpy(&inst->pros_topics_typ->config, dataset->data, dataset->size);
        }
        break;

    case EXOS_DATASET_EVENT_PUBLISHED:
        VERBOSE("dataset %s published to local server for distribution! send buffer free:%i", dataset->name, dataset->send_buffer.free);
        //handle each published dataset separately
        if(0 == strcmp(dataset->name, "odemetry"))
        {
            // ros_topic_odemety_typ *odemetry_dataset = (ros_topic_odemety_typ *)dataset->data;
        }
        break;

    case EXOS_DATASET_EVENT_DELIVERED:
        VERBOSE("dataset %s delivered to remote server for distribution! send buffer free:%i", dataset->name, dataset->send_buffer.free);
        //handle each published dataset separately
        if(0 == strcmp(dataset->name, "odemetry"))
        {
            // ros_topic_odemety_typ *odemetry_dataset = (ros_topic_odemety_typ *)dataset->data;
        }
        break;

    case EXOS_DATASET_EVENT_CONNECTION_CHANGED:
        INFO("dataset %s changed state to %s", dataset->name, exos_get_state_string(dataset->connection_state));

        switch (dataset->connection_state)
        {
        case EXOS_STATE_DISCONNECTED:
            break;
        case EXOS_STATE_CONNECTED:
            //call the dataset changed event to update the dataset when connected
            //datasetEvent(dataset,EXOS_DATASET_UPDATED,info);
            break;
        case EXOS_STATE_OPERATIONAL:
            break;
        case EXOS_STATE_ABORTED:
            ERROR("dataset %s error %d (%s) occured", dataset->name, dataset->error, exos_get_error_string(dataset->error));
            break;
        }
        break;
    }

}

static void datamodelEvent(exos_datamodel_handle_t *datamodel, const EXOS_DATAMODEL_EVENT_TYPE event_type, void *info)
{
    struct ros_topics_typCyclic *inst = (struct ros_topics_typCyclic *)datamodel->user_context;
    ros_topics_typHandle_t *handle = (ros_topics_typHandle_t *)inst->Handle;

    switch (event_type)
    {
    case EXOS_DATAMODEL_EVENT_CONNECTION_CHANGED:
        INFO("application changed state to %s", exos_get_state_string(datamodel->connection_state));

        inst->Disconnected = 0;
        inst->Connected = 0;
        inst->Operational = 0;
        inst->Aborted = 0;

        switch (datamodel->connection_state)
        {
        case EXOS_STATE_DISCONNECTED:
            inst->Disconnected = 1;
            inst->_state = 255;
            break;
        case EXOS_STATE_CONNECTED:
            inst->Connected = 1;
            break;
        case EXOS_STATE_OPERATIONAL:
            SUCCESS("ros_topics_typ operational!");
            inst->Operational = 1;
            break;
        case EXOS_STATE_ABORTED:
            ERROR("application error %d (%s) occured", datamodel->error, exos_get_error_string(datamodel->error));
            inst->_state = 255;
            inst->Aborted = 1;
            break;
        }
        break;
    case EXOS_DATAMODEL_EVENT_SYNC_STATE_CHANGED:
        break;

    default:
        break;

    }

}

_BUR_PUBLIC void ros_topics_typInit(struct ros_topics_typInit *inst)
{
    ros_topics_typHandle_t *handle;
    TMP_alloc(sizeof(ros_topics_typHandle_t), (void **)&handle);
    if (NULL == handle)
    {
        inst->Handle = 0;
        return;
    }

    memset(&handle->data, 0, sizeof(handle->data));
    handle->self = handle;

    exos_log_init(&handle->logger, "gros_topics_typ_0");

    exos_datamodel_handle_t *ros_topics_typ_datamodel = &handle->ros_topics_typ_datamodel;
    exos_dataset_handle_t *odemetry_dataset = &handle->odemetry_dataset;
    exos_dataset_handle_t *twist_dataset = &handle->twist_dataset;
    exos_dataset_handle_t *config_dataset = &handle->config_dataset;
    EXOS_ASSERT_OK(exos_datamodel_init(ros_topics_typ_datamodel, "ros_topics_typ_0", "gros_topics_typ_0"));

    EXOS_ASSERT_OK(exos_dataset_init(odemetry_dataset, ros_topics_typ_datamodel, "odemetry", &handle->data.odemetry, sizeof(handle->data.odemetry)));
    EXOS_ASSERT_OK(exos_dataset_init(twist_dataset, ros_topics_typ_datamodel, "twist", &handle->data.twist, sizeof(handle->data.twist)));
    EXOS_ASSERT_OK(exos_dataset_init(config_dataset, ros_topics_typ_datamodel, "config", &handle->data.config, sizeof(handle->data.config)));

    inst->Handle = (UDINT)handle;
}

_BUR_PUBLIC void ros_topics_typCyclic(struct ros_topics_typCyclic *inst)
{
    ros_topics_typHandle_t *handle = (ros_topics_typHandle_t *)inst->Handle;

    inst->Error = false;
    if (NULL == handle || NULL == inst->pros_topics_typ)
    {
        inst->Error = true;
        return;
    }
    if ((void *)handle != handle->self)
    {
        inst->Error = true;
        return;
    }

    ros_topics_typ *data = &handle->data;
    exos_datamodel_handle_t *ros_topics_typ_datamodel = &handle->ros_topics_typ_datamodel;
    //the user context of the datamodel points to the ros_topics_typCyclic instance
    ros_topics_typ_datamodel->user_context = inst; //set it cyclically in case the program using the FUB is retransferred
    ros_topics_typ_datamodel->user_tag = 0; //user defined
    //handle online download of the library
    if(NULL != ros_topics_typ_datamodel->datamodel_event_callback && ros_topics_typ_datamodel->datamodel_event_callback != datamodelEvent)
    {
        ros_topics_typ_datamodel->datamodel_event_callback = datamodelEvent;
        exos_log_delete(&handle->logger);
        exos_log_init(&handle->logger, "gros_topics_typ_0");
    }

    exos_dataset_handle_t *odemetry_dataset = &handle->odemetry_dataset;
    odemetry_dataset->user_context = NULL; //user defined
    odemetry_dataset->user_tag = 0; //user defined
    //handle online download of the library
    if(NULL != odemetry_dataset->dataset_event_callback && odemetry_dataset->dataset_event_callback != datasetEvent)
    {
        odemetry_dataset->dataset_event_callback = datasetEvent;
    }

    exos_dataset_handle_t *twist_dataset = &handle->twist_dataset;
    twist_dataset->user_context = NULL; //user defined
    twist_dataset->user_tag = 0; //user defined
    //handle online download of the library
    if(NULL != twist_dataset->dataset_event_callback && twist_dataset->dataset_event_callback != datasetEvent)
    {
        twist_dataset->dataset_event_callback = datasetEvent;
    }

    exos_dataset_handle_t *config_dataset = &handle->config_dataset;
    config_dataset->user_context = NULL; //user defined
    config_dataset->user_tag = 0; //user defined
    //handle online download of the library
    if(NULL != config_dataset->dataset_event_callback && config_dataset->dataset_event_callback != datasetEvent)
    {
        config_dataset->dataset_event_callback = datasetEvent;
    }

    //unregister on disable
    if (inst->_state && !inst->Enable)
    {
        inst->_state = 255;
    }

    switch (inst->_state)
    {
    case 0:
        inst->Disconnected = 1;
        inst->Connected = 0;
        inst->Operational = 0;
        inst->Aborted = 0;

        if (inst->Enable)
        {
            inst->_state = 10;
        }
        break;

    case 10:
        inst->_state = 100;

        SUCCESS("starting ros_topics_typ application..");

        //connect the datamodel, then the datasets
        EXOS_ASSERT_OK(exos_datamodel_connect_ros_topics_typ(ros_topics_typ_datamodel, datamodelEvent));
        EXOS_ASSERT_OK(exos_dataset_connect(odemetry_dataset, EXOS_DATASET_PUBLISH, datasetEvent));
        EXOS_ASSERT_OK(exos_dataset_connect(twist_dataset, EXOS_DATASET_SUBSCRIBE, datasetEvent));
        EXOS_ASSERT_OK(exos_dataset_connect(config_dataset, EXOS_DATASET_SUBSCRIBE, datasetEvent));

        inst->Active = true;
        break;

    case 100:
    case 101:
        if (inst->Start)
        {
            if (inst->_state == 100)
            {
                EXOS_ASSERT_OK(exos_datamodel_set_operational(ros_topics_typ_datamodel));
                inst->_state = 101;
            }
        }
        else
        {
            inst->_state = 100;
        }

        EXOS_ASSERT_OK(exos_datamodel_process(ros_topics_typ_datamodel));
        //put your cyclic code here!

        //publish the odemetry_dataset dataset as soon as there are changes
        if (0 != memcmp(&inst->pros_topics_typ->odemetry, &data->odemetry, sizeof(data->odemetry)))
        {
            memcpy(&data->odemetry, &inst->pros_topics_typ->odemetry, sizeof(data->odemetry));
            exos_dataset_publish(odemetry_dataset);
        }

        break;

    case 255:
        //disconnect the datamodel
        EXOS_ASSERT_OK(exos_datamodel_disconnect(ros_topics_typ_datamodel));

        inst->Active = false;
        inst->_state = 254;
        //no break

    case 254:
        if (!inst->Enable)
            inst->_state = 0;
        break;
    }

    exos_log_process(&handle->logger);

}

_BUR_PUBLIC void ros_topics_typExit(struct ros_topics_typExit *inst)
{
    ros_topics_typHandle_t *handle = (ros_topics_typHandle_t *)inst->Handle;

    if (NULL == handle)
    {
        ERROR("ros_topics_typExit: NULL handle, cannot delete resources");
        return;
    }
    if ((void *)handle != handle->self)
    {
        ERROR("ros_topics_typExit: invalid handle, cannot delete resources");
        return;
    }

    exos_datamodel_handle_t *ros_topics_typ_datamodel = &handle->ros_topics_typ_datamodel;

    EXOS_ASSERT_OK(exos_datamodel_delete(ros_topics_typ_datamodel));

    //finish with deleting the log
    exos_log_delete(&handle->logger);
    //free the allocated handle
    TMP_free(sizeof(ros_topics_typHandle_t), (void *)handle);
}
```

### Package Logical/test/ros_topics_typ/Linux - ros_topics_typ Linux resources

### exos_ros_topics_typ.h
```c
/*Automatically generated header file from ros_topics.typ*/

#ifndef _EXOS_COMP_ROS_TOPICS_TYP_H_
#define _EXOS_COMP_ROS_TOPICS_TYP_H_

#include "exos_api.h"

#if defined(_SG4)
#include <ros_topics.h>
#else
#include <stddef.h>
#include <stdint.h>
#include <stdbool.h>

typedef struct ros_config_typ
{
    double maxSpeed;
    double minSpeed;
    double baseWidth;

} ros_config_typ;

//this expresses velocity in free space broken into its linear and angular parts.
typedef struct ros_topic_vector3_typ
{
    double y;
    double z;
    double x;

} ros_topic_vector3_typ;

//This expresses velocity in free space broken into its linear and angular parts.
typedef struct ros_topic_twist_typ
{
    struct ros_topic_vector3_typ angular;
    struct ros_topic_vector3_typ linear;

} ros_topic_twist_typ;

typedef struct ros_topic_time_typ
{
    uint32_t nsec;
    uint32_t sec;

} ros_topic_time_typ;

typedef struct ros_topic_header_typ
{
    struct ros_topic_time_typ stamp;
    uint32_t seq;
    char frame_id[21];

} ros_topic_header_typ;

//This expresses velocity in free space with uncertainty.
typedef struct ros_topic_twistCor_typ
{
    struct ros_topic_twist_typ twist;

} ros_topic_twistCor_typ;

//This represents an orientation in free space in quaternion form.
typedef struct ros_topic_quaternion_typ
{
    double y;
    double z;
    double w;
    double x;

} ros_topic_quaternion_typ;

//this expresses velocity in free space broken into its linear and angular parts.
typedef struct ros_topic_point_typ
{
    double y;
    double z;
    double x;

} ros_topic_point_typ;

//A representation of pose in free space, composed of position and orientation.
typedef struct ros_topic_pose_typ
{
    struct ros_topic_point_typ position;
    struct ros_topic_quaternion_typ orientation;

} ros_topic_pose_typ;

//This represents a pose in free space with uncertainty.
typedef struct ros_topic_poseCor_typ
{
    struct ros_topic_pose_typ pose;

} ros_topic_poseCor_typ;

typedef struct ros_topic_odemety_typ
{
    struct ros_topic_poseCor_typ pose;
    struct ros_topic_twistCor_typ twist;
    struct ros_topic_header_typ header;

} ros_topic_odemety_typ;

typedef struct ros_topics_typ
{
    struct ros_topic_odemety_typ odemetry; //PUB
    struct ros_topic_twist_typ twist; //SUB
    struct ros_config_typ config; //SUB

} ros_topics_typ;

#endif // _SG4

EXOS_ERROR_CODE exos_datamodel_connect_ros_topics_typ(exos_datamodel_handle_t *datamodel, exos_datamodel_event_cb datamodel_event_callback);

#endif // _EXOS_COMP_ROS_TOPICS_TYP_H_
```

### libros_topics_typ.h
```c
#ifndef _LIBROS_TOPICS_TYP_H_
#define _LIBROS_TOPICS_TYP_H_

#include "exos_ros_topics_typ.h"

typedef void (*libros_topics_typ_event_cb)(void);
typedef void (*libros_topics_typ_method_fn)(void);
typedef int32_t (*libros_topics_typ_get_nettime_fn)(void);
typedef void (*libros_topics_typ_log_fn)(char *log_entry);

typedef struct libros_topics_typodemetry
{
    libros_topics_typ_event_cb on_change;
    int32_t nettime;
    ros_topic_odemety_typ value;
} libros_topics_typodemetry_t;

typedef struct libros_topics_typtwist
{
    libros_topics_typ_method_fn publish;
    ros_topic_twist_typ value;
} libros_topics_typtwist_t;

typedef struct libros_topics_typconfig
{
    libros_topics_typ_method_fn publish;
    ros_config_typ value;
} libros_topics_typconfig_t;

typedef struct libros_topics_typ_log
{
    libros_topics_typ_log_fn error;
    libros_topics_typ_log_fn warning;
    libros_topics_typ_log_fn success;
    libros_topics_typ_log_fn info;
    libros_topics_typ_log_fn debug;
    libros_topics_typ_log_fn verbose;
} libros_topics_typ_log_t;

typedef struct libros_topics_typ
{
    libros_topics_typ_method_fn connect;
    libros_topics_typ_method_fn disconnect;
    libros_topics_typ_method_fn process;
    libros_topics_typ_method_fn set_operational;
    libros_topics_typ_method_fn dispose;
    libros_topics_typ_get_nettime_fn get_nettime;
    libros_topics_typ_log_t log;
    libros_topics_typ_event_cb on_connected;
    libros_topics_typ_event_cb on_disconnected;
    libros_topics_typ_event_cb on_operational;
    bool is_connected;
    bool is_operational;
    libros_topics_typodemetry_t odemetry;
    libros_topics_typtwist_t twist;
    libros_topics_typconfig_t config;
} libros_topics_typ_t;

#ifdef __cplusplus
extern "C" {
#endif
libros_topics_typ_t *libros_topics_typ_init(void);
#ifdef __cplusplus
}
#endif
#endif // _LIBROS_TOPICS_TYP_H_
```
